LIN {X 0,Y 530.243,Z 390.539,A -85,B 0,C 180,E1 24517.422,E2 24517.422} C_VEL
LIN {X 0,Y 522.245,Z 380.137,A -85,B 0,C 180,E1 24516.068,E2 24516.068} C_VEL
LIN {X 0,Y 518.411,Z 375.142,A -85,B 0,C 180,E1 24515.388,E2 24515.388} C_VEL
LIN {X 0,Y 515.16,Z 370.904,A -85,B 0,C 180,E1 24514.795,E2 24514.795} C_VEL
LIN {X 0,Y 511.277,Z 366.368,A -85,B 0,C 180,E1 24514.077,E2 24514.077} C_VEL
LIN {X 0,Y 510.058,Z 364.29,A -85,B 0,C 180,E1 24513.831,E2 24513.831} C_VEL
LIN {X 0,Y 507.318,Z 361.986,A -85,B 0,C 180,E1 24513.326,E2 24513.326} C_VEL
LIN {X 0,Y 505.948,Z 358.981,A -85,B 0,C 180,E1 24513.023,E2 24513.023} C_VEL
LIN {X 0,Y 505.819,Z 358.226,A -85,B 0,C 180,E1 24512.977,E2 24512.977} C_VEL
LIN {X 0,Y 505.821,Z 358.219,A -85,B 0,C 180,E1 24509.486,E2 24509.486} C_VEL
LIN {X 0,Y 505.867,Z 358.21,A -85,B 0,C 180,E1 24506.154,E2 24506.154} C_VEL
LIN {X 0,Y 505.817,Z 358.219,A -85,B 0,C 180,E1 24502.796,E2 24502.796} C_VEL
LIN {X 0,Y 505.818,Z 358.222,A -85,B 0,C 180,E1 24499.276,E2 24499.276} C_VEL
LIN {X 0,Y 505.867,Z 358.218,A -85,B 0,C 180,E1 24495.829,E2 24495.829} C_VEL
LIN {X 0,Y 505.827,Z 358.218,A -85,B 0,C 180,E1 24492.443,E2 24492.443} C_VEL
LIN {X 0,Y 505.81,Z 358.211,A -85,B 0,C 180,E1 24488.985,E2 24488.985} C_VEL
LIN {X 0,Y 505.861,Z 358.197,A -85,B 0,C 180,E1 24485.672,E2 24485.672} C_VEL
LIN {X 0,Y 505.825,Z 358.208,A -85,B 0,C 180,E1 24482.266,E2 24482.266} C_VEL
LIN {X 0,Y 505.814,Z 358.223,A -85,B 0,C 180,E1 24478.867,E2 24478.867} C_VEL
LIN {X 0,Y 505.86,Z 358.216,A -85,B 0,C 180,E1 24475.465,E2 24475.465} C_VEL
LIN {X 0,Y 505.819,Z 358.203,A -85,B 0,C 180,E1 24472.161,E2 24472.161} C_VEL
LIN {X 0,Y 505.809,Z 358.199,A -85,B 0,C 180,E1 24468.666,E2 24468.666} C_VEL
LIN {X 0,Y 505.856,Z 358.198,A -85,B 0,C 180,E1 24465.227,E2 24465.227} C_VEL
LIN {X 0,Y 505.836,Z 358.211,A -85,B 0,C 180,E1 24461.801,E2 24461.801} C_VEL
LIN {X 0,Y 505.811,Z 358.223,A -85,B 0,C 180,E1 24458.427,E2 24458.427} C_VEL
LIN {X 0,Y 505.86,Z 358.216,A -85,B 0,C 180,E1 24455.101,E2 24455.101} C_VEL
LIN {X 0,Y 505.833,Z 358.216,A -85,B 0,C 180,E1 24451.679,E2 24451.679} C_VEL
LIN {X 0,Y 505.809,Z 358.224,A -85,B 0,C 180,E1 24448.215,E2 24448.215} C_VEL
LIN {X 0,Y 505.856,Z 358.329,A -85,B 0,C 180,E1 24446.764,E2 24446.764} C_VEL
LIN {X 0,Y 507.026,Z 361.574,A -85,B 0,C 180,E1 24446.076,E2 24446.076} C_VEL
LIN {X 0,Y 508.127,Z 363.457,A -85,B 0,C 180,E1 24445.614,E2 24445.614} C_VEL
LIN {X 0,Y 511.472,Z 370.526,A -85,B 0,C 180,E1 24444.127,E2 24444.127} C_VEL
LIN {X 0,Y 517.191,Z 378.321,A -85,B 0,C 180,E1 24443.057,E2 24443.057} C_VEL
LIN {X 0,Y 526.687,Z 391.502,A -85,B 0,C 180,E1 24441.382,E2 24441.382} C_VEL
LIN {X 0,Y 538.736,Z 409.397,A -85,B 0,C 180,E1 24439.401,E2 24439.401} C_VEL
LIN {X 0,Y 550.421,Z 428.049,A -85,B 0,C 180,E1 24437.609,E2 24437.609} C_VEL
LIN {X 0,Y 559.833,Z 444.357,A -85,B 0,C 180,E1 24436.239,E2 24436.239} C_VEL
LIN {X 0,Y 551.218,Z 697.847,A -85,B 0,C 180,E1 24432.584,E2 24432.584} C_VEL
LIN {X 0,Y 548.851,Z 765.211,A -85,B 0,C 180,E1 24431.594,E2 24431.594} C_VEL
LIN {X 0,Y 546.947,Z 790.534,A -85,B 0,C 180,E1 24431.062,E2 24431.062} C_VEL
LIN {X 0,Y 544.812,Z 812.3,A -85,B 0,C 180,E1 24430.449,E2 24430.449} C_VEL
LIN {X 0,Y 541.812,Z 837.253,A -85,B 0,C 180,E1 24429.545,E2 24429.545} C_VEL
LIN {X 0,Y 538.992,Z 857.715,A -85,B 0,C 180,E1 24428.627,E2 24428.627} C_VEL
LIN {X 0,Y 535.358,Z 881.083,A -85,B 0,C 180,E1 24427.373,E2 24427.373} C_VEL
LIN {X 0,Y 532.124,Z 900.104,A -85,B 0,C 180,E1 24426.159,E2 24426.159} C_VEL
LIN {X 0,Y 528.453,Z 920.63,A -85,B 0,C 180,E1 24424.651,E2 24424.651} C_VEL
LIN {X 0,Y 524.681,Z 940.175,A -85,B 0,C 180,E1 24422.962,E2 24422.962} C_VEL
LIN {X 0,Y 521.204,Z 958.071,A -85,B 0,C 180,E1 24421.196,E2 24421.196} C_VEL
LIN {X 0,Y 517.662,Z 976.147,A -85,B 0,C 180,E1 24419.127,E2 24419.127} C_VEL
LIN {X 0,Y 514.766,Z 991.223,A -85,B 0,C 180,E1 24417.159,E2 24417.159} C_VEL
LIN {X 0,Y 511.753,Z 1007.595,A -85,B 0,C 180,E1 24414.695,E2 24414.695} C_VEL
LIN {X 0,Y 509.578,Z 1020.26,A -85,B 0,C 180,E1 24412.497,E2 24412.497} C_VEL
LIN {X 0,Y 507.526,Z 1033.62,A -85,B 0,C 180,E1 24409.808,E2 24409.808} C_VEL
LIN {X 0,Y 506.184,Z 1043.698,A -85,B 0,C 180,E1 24407.427,E2 24407.427} C_VEL
LIN {X 0,Y 505.112,Z 1053.565,A -85,B 0,C 180,E1 24404.678,E2 24404.678} C_VEL
LIN {X 0,Y 504.506,Z 1060.698,A -85,B 0,C 180,E1 24402.243,E2 24402.243} C_VEL
LIN {X 0,Y 504.146,Z 1066.814,A -85,B 0,C 180,E1 24399.693,E2 24399.693} C_VEL
LIN {X 0,Y 503.971,Z 1071.694,A -85,B 0,C 180,E1 24396.951,E2 24396.951} C_VEL
LIN {X 0,Y 503.931,Z 1074.534,A -85,B 0,C 180,E1 24394.666,E2 24394.666} C_VEL
LIN {X 0,Y 503.925,Z 1076.418,A -85,B 0,C 180,E1 24392.161,E2 24392.161} C_VEL
LIN {X 0,Y 503.916,Z 1076.851,A -85,B 0,C 180,E1 24389.432,E2 24389.432} C_VEL
LIN {X 0,Y 503.926,Z 1076.004,A -85,B 0,C 180,E1 24387.157,E2 24387.157} C_VEL
LIN {X 0,Y 503.939,Z 1073.839,A -85,B 0,C 180,E1 24384.649,E2 24384.649} C_VEL
LIN {X 0,Y 504.022,Z 1069.764,A -85,B 0,C 180,E1 24381.863,E2 24381.863} C_VEL
LIN {X 0,Y 504.23,Z 1064.959,A -85,B 0,C 180,E1 24379.488,E2 24379.488} C_VEL
LIN {X 0,Y 504.701,Z 1058.167,A -85,B 0,C 180,E1 24376.831,E2 24376.831} C_VEL
LIN {X 0,Y 505.456,Z 1049.904,A -85,B 0,C 180,E1 24374.276,E2 24374.276} C_VEL
LIN {X 0,Y 506.477,Z 1041.045,A -85,B 0,C 180,E1 24371.944,E2 24371.944} C_VEL
LIN {X 0,Y 508.133,Z 1028.955,A -85,B 0,C 180,E1 24369.256,E2 24369.256} C_VEL
LIN {X 0,Y 509.968,Z 1017.316,A -85,B 0,C 180,E1 24367.034,E2 24367.034} C_VEL
LIN {X 0,Y 512.628,Z 1001.746,A -85,B 0,C 180,E1 24364.465,E2 24364.465} C_VEL
LIN {X 0,Y 515.141,Z 987.899,A -85,B 0,C 180,E1 24362.486,E2 24362.486} C_VEL
LIN {X 0,Y 518.363,Z 970.778,A -85,B 0,C 180,E1 24360.333,E2 24360.333} C_VEL
LIN {X 0,Y 521.652,Z 953.358,A -85,B 0,C 180,E1 24358.448,E2 24358.448} C_VEL
LIN {X 0,Y 525.288,Z 934.182,A -85,B 0,C 180,E1 24356.625,E2 24356.625} C_VEL
LIN {X 0,Y 528.894,Z 913.938,A -85,B 0,C 180,E1 24354.986,E2 24354.986} C_VEL
LIN {X 0,Y 532.482,Z 893.313,A -85,B 0,C 180,E1 24353.536,E2 24353.536} C_VEL
LIN {X 0,Y 535.856,Z 871.76,A -85,B 0,C 180,E1 24352.263,E2 24352.263} C_VEL
LIN {X 0,Y 539.01,Z 850.159,A -85,B 0,C 180,E1 24351.181,E2 24351.181} C_VEL
LIN {X 0,Y 541.922,Z 826.849,A -85,B 0,C 180,E1 24350.224,E2 24350.224} C_VEL
LIN {X 0,Y 544.113,Z 806.615,A -85,B 0,C 180,E1 24349.551,E2 24349.551} C_VEL
LIN {X 0,Y 546.315,Z 781.962,A -85,B 0,C 180,E1 24348.911,E2 24348.911} C_VEL
LIN {X 0,Y 547.686,Z 758.897,A -85,B 0,C 180,E1 24348.481,E2 24348.481} C_VEL
LIN {X 0,Y 555.231,Z 521.007,A -85,B 0,C 180,E1 24345.07,E2 24345.07} C_VEL
LIN {X 0,Y 557.675,Z 443.181,A -85,B 0,C 180,E1 24343.938,E2 24343.938} C_VEL
LIN {X 0,Y 544.63,Z 420.749,A -85,B 0,C 180,E1 24342.125,E2 24342.125} C_VEL
LIN {X 0,Y 532.554,Z 401.419,A -85,B 0,C 180,E1 24340.338,E2 24340.338} C_VEL
LIN {X 0,Y 522.976,Z 387.268,A -85,B 0,C 180,E1 24338.838,E2 24338.838} C_VEL
LIN {X 0,Y 514.362,Z 375.002,A -85,B 0,C 180,E1 24337.408,E2 24337.408} C_VEL
LIN {X 0,Y 511.191,Z 370.226,A -85,B 0,C 180,E1 24336.835,E2 24336.835} C_VEL
LIN {X 0,Y 507.157,Z 361.687,A -85,B 0,C 180,E1 24335.095,E2 24335.095} C_VEL
LIN {X 0,Y 505.824,Z 358.204,A -85,B 0,C 180,E1 24334.358,E2 24334.358} C_VEL
LIN {X 0,Y 505.852,Z 358.197,A -85,B 0,C 180,E1 24331.058,E2 24331.058} C_VEL
LIN {X 0,Y 505.811,Z 358.2,A -85,B 0,C 180,E1 24327.674,E2 24327.674} C_VEL
LIN {X 0,Y 505.823,Z 358.203,A -85,B 0,C 180,E1 24324.154,E2 24324.154} C_VEL
LIN {X 0,Y 505.861,Z 358.219,A -85,B 0,C 180,E1 24320.842,E2 24320.842} C_VEL
LIN {X 0,Y 505.814,Z 358.22,A -85,B 0,C 180,E1 24317.367,E2 24317.367} C_VEL
LIN {X 0,Y 505.814,Z 358.199,A -85,B 0,C 180,E1 24313.839,E2 24313.839} C_VEL
LIN {X 0,Y 505.862,Z 358.197,A -85,B 0,C 180,E1 24310.477,E2 24310.477} C_VEL
LIN {X 0,Y 505.823,Z 358.222,A -85,B 0,C 180,E1 24307.04,E2 24307.04} C_VEL
LIN {X 0,Y 505.81,Z 358.202,A -85,B 0,C 180,E1 24303.513,E2 24303.513} C_VEL
LIN {X 0,Y 505.858,Z 358.193,A -85,B 0,C 180,E1 24300.113,E2 24300.113} C_VEL
LIN {X 0,Y 505.833,Z 358.221,A -85,B 0,C 180,E1 24296.714,E2 24296.714} C_VEL
LIN {X 0,Y 505.808,Z 358.199,A -85,B 0,C 180,E1 24293.302,E2 24293.302} C_VEL
LIN {X 0,Y 505.858,Z 358.198,A -85,B 0,C 180,E1 24289.983,E2 24289.983} C_VEL
LIN {X 0,Y 505.837,Z 358.22,A -85,B 0,C 180,E1 24286.511,E2 24286.511} C_VEL
LIN {X 0,Y 505.811,Z 358.202,A -85,B 0,C 180,E1 24283.092,E2 24283.092} C_VEL
LIN {X 0,Y 505.858,Z 358.195,A -85,B 0,C 180,E1 24279.763,E2 24279.763} C_VEL
LIN {X 0,Y 505.829,Z 358.223,A -85,B 0,C 180,E1 24276.465,E2 24276.465} C_VEL
LIN {X 0,Y 505.815,Z 358.223,A -85,B 0,C 180,E1 24272.957,E2 24272.957} C_VEL
LIN {X 0,Y 505.863,Z 358.201,A -85,B 0,C 180,E1 24269.601,E2 24269.601} C_VEL
LIN {X 0,Y 505.831,Z 358.202,A -85,B 0,C 180,E1 24266.257,E2 24266.257} C_VEL
LIN {X 0,Y 505.814,Z 358.208,A -85,B 0,C 180,E1 24262.778,E2 24262.778} C_VEL
LIN {X 0,Y 505.887,Z 358.359,A -85,B 0,C 180,E1 24261.782,E2 24261.782} C_VEL
LIN {X 0,Y 507.038,Z 361.49,A -85,B 0,C 180,E1 24261.537,E2 24261.537} C_VEL
LIN {X 0,Y 509.577,Z 364.042,A -85,B 0,C 180,E1 24261.104,E2 24261.104} C_VEL
LIN {X 0,Y 510.514,Z 365.429,A -85,B 0,C 180,E1 24260.936,E2 24260.936} C_VEL
LIN {X 0,Y 513.243,Z 369.092,A -85,B 0,C 180,E1 24260.463,E2 24260.463} C_VEL
LIN {X 0,Y 514.716,Z 370.731,A -85,B 0,C 180,E1 24260.219,E2 24260.219} C_VEL
LIN {X 0,Y 517.989,Z 375.01,A -85,B 0,C 180,E1 24259.673,E2 24259.673} C_VEL
LIN {X 0,Y 531.008,Z 392.505,A -85,B 0,C 180,E1 24257.614,E2 24257.614} C_VEL
LIN {X 0,Y 543.149,Z 409.924,A -85,B 0,C 180,E1 24255.83,E2 24255.83} C_VEL
LIN {X 0,Y 556.689,Z 432.23,A -85,B 0,C 180,E1 24253.943,E2 24253.943} C_VEL
LIN {X 0,Y 557.876,Z 434.704,A -85,B 0,C 180,E1 24253.775,E2 24253.775} C_VEL
LIN {X 0,Y 549.924,Z 680.488,A -85,B 0,C 180,E1 24250.254,E2 24250.254} C_VEL
LIN {X 0,Y 547.775,Z 743.673,A -85,B 0,C 180,E1 24249.329,E2 24249.329} C_VEL
LIN {X 0,Y 546.096,Z 768.42,A -85,B 0,C 180,E1 24248.795,E2 24248.795} C_VEL
LIN {X 0,Y 544.147,Z 790.154,A -85,B 0,C 180,E1 24248.172,E2 24248.172} C_VEL
LIN {X 0,Y 541.471,Z 814.447,A -85,B 0,C 180,E1 24247.278,E2 24247.278} C_VEL
LIN {X 0,Y 538.798,Z 834.992,A -85,B 0,C 180,E1 24246.35,E2 24246.35} C_VEL
LIN {X 0,Y 535.419,Z 857.913,A -85,B 0,C 180,E1 24245.113,E2 24245.113} C_VEL
LIN {X 0,Y 535.072,Z 860.018,A -85,B 0,C 180,E1 24244.984,E2 24244.984} C_VEL
LIN {X 0,Y 533.151,Z 866.91,A -85,B 0,C 180,E1 24244.627,E2 24244.627} C_VEL
LIN {X 0,Y 525.296,Z 883.992,A -85,B 0,C 180,E1 24243.86,E2 24243.86} C_VEL
LIN {X 0,Y 523.292,Z 890.316,A -85,B 0,C 180,E1 24243.44,E2 24243.44} C_VEL
LIN {X 0,Y 519.831,Z 908.643,A -85,B 0,C 180,E1 24241.935,E2 24241.935} C_VEL
LIN {X 0,Y 515.922,Z 928.193,A -85,B 0,C 180,E1 24240.069,E2 24240.069} C_VEL
LIN {X 0,Y 512.604,Z 944.372,A -85,B 0,C 180,E1 24238.294,E2 24238.294} C_VEL
LIN {X 0,Y 508.891,Z 962.559,A -85,B 0,C 180,E1 24235.986,E2 24235.986} C_VEL
LIN {X 0,Y 506.164,Z 976.066,A -85,B 0,C 180,E1 24234.013,E2 24234.013} C_VEL
LIN {X 0,Y 503.35,Z 990.707,A -85,B 0,C 180,E1 24231.561,E2 24231.561} C_VEL
LIN {X 0,Y 501.164,Z 1002.678,A -85,B 0,C 180,E1 24229.22,E2 24229.22} C_VEL
LIN {X 0,Y 499.344,Z 1014.112,A -85,B 0,C 180,E1 24226.639,E2 24226.639} C_VEL
LIN {X 0,Y 497.986,Z 1023.606,A -85,B 0,C 180,E1 24224.061,E2 24224.061} C_VEL
LIN {X 0,Y 497.066,Z 1031.627,A -85,B 0,C 180,E1 24221.487,E2 24221.487} C_VEL
LIN {X 0,Y 496.434,Z 1038.548,A -85,B 0,C 180,E1 24218.688,E2 24218.688} C_VEL
LIN {X 0,Y 496.146,Z 1043.064,A -85,B 0,C 180,E1 24216.364,E2 24216.364} C_VEL
LIN {X 0,Y 495.985,Z 1047.067,A -85,B 0,C 180,E1 24213.583,E2 24213.583} C_VEL
LIN {X 0,Y 495.938,Z 1049.294,A -85,B 0,C 180,E1 24210.924,E2 24210.924} C_VEL
LIN {X 0,Y 495.918,Z 1050.148,A -85,B 0,C 180,E1 24208.614,E2 24208.614} C_VEL
LIN {X 0,Y 495.936,Z 1049.805,A -85,B 0,C 180,E1 24205.838,E2 24205.838} C_VEL
LIN {X 0,Y 495.968,Z 1048.022,A -85,B 0,C 180,E1 24203.285,E2 24203.285} C_VEL
LIN {X 0,Y 496.06,Z 1045.155,A -85,B 0,C 180,E1 24200.837,E2 24200.837} C_VEL
LIN {X 0,Y 496.332,Z 1040.111,A -85,B 0,C 180,E1 24197.906,E2 24197.906} C_VEL
LIN {X 0,Y 496.805,Z 1034.416,A -85,B 0,C 180,E1 24195.429,E2 24195.429} C_VEL
LIN {X 0,Y 497.664,Z 1026.716,A -85,B 0,C 180,E1 24192.701,E2 24192.701} C_VEL
LIN {X 0,Y 498.91,Z 1017.376,A -85,B 0,C 180,E1 24190.043,E2 24190.043} C_VEL
LIN {X 0,Y 500.649,Z 1006.723,A -85,B 0,C 180,E1 24187.452,E2 24187.452} C_VEL
LIN {X 0,Y 502.833,Z 994.441,A -85,B 0,C 180,E1 24184.941,E2 24184.941} C_VEL
LIN {X 0,Y 505.349,Z 981.711,A -85,B 0,C 180,E1 24182.673,E2 24182.673} C_VEL
LIN {X 0,Y 508.518,Z 966.224,A -85,B 0,C 180,E1 24180.297,E2 24180.297} C_VEL
LIN {X 0,Y 511.718,Z 951.187,A -85,B 0,C 180,E1 24178.29,E2 24178.29} C_VEL
LIN {X 0,Y 515.692,Z 932.365,A -85,B 0,C 180,E1 24176.114,E2 24176.114} C_VEL
LIN {X 0,Y 519.195,Z 915.589,A -85,B 0,C 180,E1 24174.436,E2 24174.436} C_VEL
LIN {X 0,Y 523.484,Z 894.286,A -85,B 0,C 180,E1 24172.598,E2 24172.598} C_VEL
LIN {X 0,Y 526.959,Z 875.808,A -85,B 0,C 180,E1 24171.232,E2 24171.232} C_VEL
LIN {X 0,Y 530.668,Z 854.628,A -85,B 0,C 180,E1 24169.879,E2 24169.879} C_VEL
LIN {X 0,Y 533.938,Z 833.645,A -85,B 0,C 180,E1 24168.763,E2 24168.763} C_VEL
LIN {X 0,Y 537.103,Z 810.848,A -85,B 0,C 180,E1 24167.738,E2 24167.738} C_VEL
LIN {X 0,Y 539.796,Z 787.034,A -85,B 0,C 180,E1 24166.895,E2 24166.895} C_VEL
LIN {X 0,Y 542.027,Z 763.422,A -85,B 0,C 180,E1 24166.239,E2 24166.239} C_VEL
LIN {X 0,Y 543.601,Z 738.929,A -85,B 0,C 180,E1 24165.755,E2 24165.755} C_VEL
LIN {X 0,Y 552.114,Z 499.336,A -85,B 0,C 180,E1 24162.264,E2 24162.264} C_VEL
LIN {X 0,Y 554.239,Z 438.354,A -85,B 0,C 180,E1 24161.36,E2 24161.36} C_VEL
LIN {X 0,Y 541.092,Z 417.091,A -85,B 0,C 180,E1 24159.385,E2 24159.385} C_VEL
LIN {X 0,Y 530.106,Z 401.533,A -85,B 0,C 180,E1 24157.637,E2 24157.637} C_VEL
LIN {X 0,Y 519.296,Z 387.153,A -85,B 0,C 180,E1 24155.793,E2 24155.793} C_VEL
LIN {X 0,Y 514.694,Z 381.339,A -85,B 0,C 180,E1 24154.966,E2 24154.966} C_VEL
LIN {X 0,Y 510.833,Z 376.392,A -85,B 0,C 180,E1 24154.246,E2 24154.246} C_VEL
LIN {X 0,Y 507.61,Z 372.243,A -85,B 0,C 180,E1 24153.626,E2 24153.626} C_VEL
LIN {X 0,Y 506.536,Z 370.989,A -85,B 0,C 180,E1 24153.418,E2 24153.418} C_VEL
LIN {X 0,Y 503.64,Z 367.828,A -85,B 0,C 180,E1 24152.854,E2 24152.854} C_VEL
LIN {X 0,Y 502.365,Z 365.417,A -85,B 0,C 180,E1 24152.575,E2 24152.575} C_VEL
LIN {X 0,Y 499.464,Z 363.017,A -85,B 0,C 180,E1 24152.006,E2 24152.006} C_VEL
LIN {X 0,Y 498.07,Z 360.156,A -85,B 0,C 180,E1 24151.683,E2 24151.683} C_VEL
LIN {X 0,Y 497.886,Z 359.196,A -85,B 0,C 180,E1 24151.612,E2 24151.612} C_VEL
LIN {X 0,Y 497.942,Z 359.189,A -85,B 0,C 180,E1 24148.172,E2 24148.172} C_VEL
LIN {X 0,Y 497.886,Z 359.195,A -85,B 0,C 180,E1 24144.691,E2 24144.691} C_VEL
LIN {X 0,Y 497.874,Z 359.195,A -85,B 0,C 180,E1 24141.192,E2 24141.192} C_VEL
LIN {X 0,Y 497.913,Z 359.189,A -85,B 0,C 180,E1 24137.773,E2 24137.773} C_VEL
LIN {X 0,Y 497.889,Z 359.193,A -85,B 0,C 180,E1 24134.42,E2 24134.42} C_VEL
LIN {X 0,Y 497.873,Z 359.204,A -85,B 0,C 180,E1 24130.999,E2 24130.999} C_VEL
LIN {X 0,Y 497.92,Z 359.208,A -85,B 0,C 180,E1 24127.616,E2 24127.616} C_VEL
LIN {X 0,Y 497.899,Z 359.204,A -85,B 0,C 180,E1 24124.146,E2 24124.146} C_VEL
LIN {X 0,Y 497.869,Z 359.195,A -85,B 0,C 180,E1 24120.69,E2 24120.69} C_VEL
LIN {X 0,Y 497.905,Z 359.186,A -85,B 0,C 180,E1 24117.353,E2 24117.353} C_VEL
LIN {X 0,Y 497.906,Z 359.195,A -85,B 0,C 180,E1 24113.89,E2 24113.89} C_VEL
LIN {X 0,Y 497.871,Z 359.213,A -85,B 0,C 180,E1 24110.521,E2 24110.521} C_VEL
LIN {X 0,Y 497.892,Z 359.209,A -85,B 0,C 180,E1 24107.002,E2 24107.002} C_VEL
LIN {X 0,Y 497.908,Z 359.189,A -85,B 0,C 180,E1 24103.671,E2 24103.671} C_VEL
LIN {X 0,Y 497.868,Z 359.188,A -85,B 0,C 180,E1 24100.281,E2 24100.281} C_VEL
LIN {X 0,Y 497.89,Z 359.187,A -85,B 0,C 180,E1 24096.82,E2 24096.82} C_VEL
LIN {X 0,Y 497.924,Z 359.186,A -85,B 0,C 180,E1 24093.331,E2 24093.331} C_VEL
LIN {X 0,Y 497.876,Z 359.211,A -85,B 0,C 180,E1 24089.949,E2 24089.949} C_VEL
LIN {X 0,Y 497.886,Z 359.31,A -85,B 0,C 180,E1 24088.023,E2 24088.023} C_VEL
LIN {X 0,Y 499.189,Z 362.632,A -85,B 0,C 180,E1 24087.26,E2 24087.26} C_VEL
LIN {X 0,Y 500.218,Z 364.49,A -85,B 0,C 180,E1 24086.79,E2 24086.79} C_VEL
LIN {X 0,Y 502.776,Z 369.865,A -85,B 0,C 180,E1 24085.577,E2 24085.577} C_VEL
LIN {X 0,Y 513.514,Z 384.325,A -85,B 0,C 180,E1 24083.48,E2 24083.48} C_VEL
LIN {X 0,Y 523.228,Z 398.04,A -85,B 0,C 180,E1 24081.727,E2 24081.727} C_VEL
LIN {X 0,Y 534.82,Z 415.4,A -85,B 0,C 180,E1 24079.781,E2 24079.781} C_VEL
LIN {X 0,Y 546.385,Z 434.053,A -85,B 0,C 180,E1 24077.969,E2 24077.969} C_VEL
LIN {X 0,Y 554.244,Z 447.991,A -85,B 0,C 180,E1 24076.792,E2 24076.792} C_VEL
LIN {X 0,Y 545.342,Z 699.596,A -85,B 0,C 180,E1 24073.135,E2 24073.135} C_VEL
LIN {X 0,Y 542.94,Z 765.137,A -85,B 0,C 180,E1 24072.163,E2 24072.163} C_VEL
LIN {X 0,Y 540.977,Z 790.404,A -85,B 0,C 180,E1 24071.628,E2 24071.628} C_VEL
LIN {X 0,Y 538.79,Z 811.938,A -85,B 0,C 180,E1 24071.02,E2 24071.02} C_VEL
LIN {X 0,Y 535.62,Z 837.328,A -85,B 0,C 180,E1 24070.094,E2 24070.094} C_VEL
LIN {X 0,Y 532.72,Z 857.586,A -85,B 0,C 180,E1 24069.178,E2 24069.178} C_VEL
LIN {X 0,Y 528.916,Z 881.067,A -85,B 0,C 180,E1 24067.908,E2 24067.908} C_VEL
LIN {X 0,Y 525.437,Z 900.712,A -85,B 0,C 180,E1 24066.639,E2 24066.639} C_VEL
LIN {X 0,Y 521.595,Z 921.255,A -85,B 0,C 180,E1 24065.106,E2 24065.106} C_VEL
LIN {X 0,Y 517.677,Z 940.697,A -85,B 0,C 180,E1 24063.4,E2 24063.4} C_VEL
LIN {X 0,Y 513.853,Z 959.576,A -85,B 0,C 180,E1 24061.504,E2 24061.504} C_VEL
LIN {X 0,Y 510.258,Z 976.954,A -85,B 0,C 180,E1 24059.463,E2 24059.463} C_VEL
LIN {X 0,Y 506.928,Z 993.639,A -85,B 0,C 180,E1 24057.233,E2 24057.233} C_VEL
LIN {X 0,Y 503.991,Z 1008.732,A -85,B 0,C 180,E1 24054.872,E2 24054.872} C_VEL
LIN {X 0,Y 501.516,Z 1022.662,A -85,B 0,C 180,E1 24052.383,E2 24052.383} C_VEL
LIN {X 0,Y 499.522,Z 1035.008,A -85,B 0,C 180,E1 24049.773,E2 24049.773} C_VEL
LIN {X 0,Y 498.083,Z 1045.661,A -85,B 0,C 180,E1 24047.163,E2 24047.163} C_VEL
LIN {X 0,Y 497.047,Z 1054.808,A -85,B 0,C 180,E1 24044.445,E2 24044.445} C_VEL
LIN {X 0,Y 496.461,Z 1061.733,A -85,B 0,C 180,E1 24041.973,E2 24041.973} C_VEL
LIN {X 0,Y 496.072,Z 1068.23,A -85,B 0,C 180,E1 24039.012,E2 24039.012} C_VEL
LIN {X 0,Y 495.952,Z 1072.14,A -85,B 0,C 180,E1 24036.599,E2 24036.599} C_VEL
LIN {X 0,Y 495.92,Z 1075.135,A -85,B 0,C 180,E1 24033.931,E2 24033.931} C_VEL
LIN {X 0,Y 495.924,Z 1076.499,A -85,B 0,C 180,E1 24031.271,E2 24031.271} C_VEL
LIN {X 0,Y 495.93,Z 1076.545,A -85,B 0,C 180,E1 24028.96,E2 24028.96} C_VEL
LIN {X 0,Y 495.924,Z 1075.362,A -85,B 0,C 180,E1 24026.405,E2 24026.405} C_VEL
LIN {X 0,Y 495.952,Z 1072.445,A -85,B 0,C 180,E1 24023.634,E2 24023.634} C_VEL
LIN {X 0,Y 496.055,Z 1068.768,A -85,B 0,C 180,E1 24021.305,E2 24021.305} C_VEL
LIN {X 0,Y 496.357,Z 1063.169,A -85,B 0,C 180,E1 24018.614,E2 24018.614} C_VEL
LIN {X 0,Y 496.943,Z 1055.708,A -85,B 0,C 180,E1 24015.89,E2 24015.89} C_VEL
LIN {X 0,Y 497.799,Z 1047.592,A -85,B 0,C 180,E1 24013.428,E2 24013.428} C_VEL
LIN {X 0,Y 499.241,Z 1036.445,A -85,B 0,C 180,E1 24010.619,E2 24010.619} C_VEL
LIN {X 0,Y 500.875,Z 1025.768,A -85,B 0,C 180,E1 24008.327,E2 24008.327} C_VEL
LIN {X 0,Y 503.406,Z 1010.951,A -85,B 0,C 180,E1 24005.598,E2 24005.598} C_VEL
LIN {X 0,Y 505.876,Z 997.537,A -85,B 0,C 180,E1 24003.468,E2 24003.468} C_VEL
LIN {X 0,Y 509.269,Z 980.036,A -85,B 0,C 180,E1 24001.055,E2 24001.055} C_VEL
LIN {X 0,Y 512.399,Z 964.186,A -85,B 0,C 180,E1 23999.162,E2 23999.162} C_VEL
LIN {X 0,Y 516.202,Z 944.946,A -85,B 0,C 180,E1 23997.155,E2 23997.155} C_VEL
LIN {X 0,Y 519.647,Z 927.057,A -85,B 0,C 180,E1 23995.549,E2 23995.549} C_VEL
LIN {X 0,Y 523.461,Z 906.852,A -85,B 0,C 180,E1 23993.962,E2 23993.962} C_VEL
LIN {X 0,Y 527.087,Z 885.661,A -85,B 0,C 180,E1 23992.556,E2 23992.556} C_VEL
LIN {X 0,Y 530.399,Z 865.227,A -85,B 0,C 180,E1 23991.392,E2 23991.392} C_VEL
LIN {X 0,Y 533.687,Z 841.975,A -85,B 0,C 180,E1 23990.292,E2 23990.292} C_VEL
LIN {X 0,Y 536.298,Z 821.174,A -85,B 0,C 180,E1 23989.482,E2 23989.482} C_VEL
LIN {X 0,Y 539.015,Z 795.008,A -85,B 0,C 180,E1 23988.68,E2 23988.68} C_VEL
LIN {X 0,Y 540.805,Z 772.952,A -85,B 0,C 180,E1 23988.178,E2 23988.178} C_VEL
LIN {X 0,Y 542.31,Z 740.397,A -85,B 0,C 180,E1 23987.651,E2 23987.651} C_VEL
LIN {X 0,Y 550.562,Z 489.738,A -85,B 0,C 180,E1 23984.039,E2 23984.039} C_VEL
LIN {X 0,Y 551.919,Z 446.519,A -85,B 0,C 180,E1 23983.397,E2 23983.397} C_VEL
LIN {X 0,Y 538.465,Z 423.266,A -85,B 0,C 180,E1 23981.47,E2 23981.47} C_VEL
LIN {X 0,Y 525.532,Z 402.827,A -85,B 0,C 180,E1 23979.491,E2 23979.491} C_VEL
LIN {X 0,Y 514.351,Z 386.33,A -85,B 0,C 180,E1 23977.655,E2 23977.655} C_VEL
LIN {X 0,Y 506.757,Z 375.71,A -85,B 0,C 180,E1 23976.33,E2 23976.33} C_VEL
LIN {X 0,Y 502.476,Z 369.783,A -85,B 0,C 180,E1 23975.523,E2 23975.523} C_VEL
LIN {X 0,Y 500.933,Z 366.363,A -85,B 0,C 180,E1 23974.811,E2 23974.811} C_VEL
LIN {X 0,Y 499.417,Z 363.014,A -85,B 0,C 180,E1 23974.097,E2 23974.097} C_VEL
LIN {X 0,Y 497.934,Z 359.493,A -85,B 0,C 180,E1 23973.347,E2 23973.347} C_VEL
LIN {X 0,Y 497.913,Z 359.2,A -85,B 0,C 180,E1 23973.108,E2 23973.108} C_VEL
LIN {X 0,Y 497.87,Z 359.203,A -85,B 0,C 180,E1 23969.74,E2 23969.74} C_VEL
LIN {X 0,Y 497.897,Z 359.191,A -85,B 0,C 180,E1 23966.348,E2 23966.348} C_VEL
LIN {X 0,Y 497.914,Z 359.181,A -85,B 0,C 180,E1 23962.929,E2 23962.929} C_VEL
LIN {X 0,Y 497.868,Z 359.19,A -85,B 0,C 180,E1 23959.597,E2 23959.597} C_VEL
LIN {X 0,Y 497.892,Z 359.206,A -85,B 0,C 180,E1 23956.09,E2 23956.09} C_VEL
LIN {X 0,Y 497.913,Z 359.2,A -85,B 0,C 180,E1 23952.762,E2 23952.762} C_VEL
LIN {X 0,Y 497.868,Z 359.182,A -85,B 0,C 180,E1 23949.362,E2 23949.362} C_VEL
LIN {X 0,Y 497.889,Z 359.199,A -85,B 0,C 180,E1 23945.879,E2 23945.879} C_VEL
LIN {X 0,Y 497.923,Z 359.202,A -85,B 0,C 180,E1 23942.417,E2 23942.417} C_VEL
LIN {X 0,Y 497.871,Z 359.179,A -85,B 0,C 180,E1 23939.079,E2 23939.079} C_VEL
LIN {X 0,Y 497.877,Z 359.202,A -85,B 0,C 180,E1 23935.508,E2 23935.508} C_VEL
LIN {X 0,Y 497.925,Z 359.201,A -85,B 0,C 180,E1 23932.035,E2 23932.035} C_VEL
LIN {X 0,Y 497.896,Z 359.177,A -85,B 0,C 180,E1 23928.526,E2 23928.526} C_VEL
LIN {X 0,Y 497.872,Z 359.2,A -85,B 0,C 180,E1 23925.104,E2 23925.104} C_VEL
LIN {X 0,Y 497.905,Z 359.211,A -85,B 0,C 180,E1 23921.622,E2 23921.622} C_VEL
LIN {X 0,Y 497.915,Z 359.186,A -85,B 0,C 180,E1 23918.191,E2 23918.191} C_VEL
LIN {X 0,Y 497.873,Z 359.185,A -85,B 0,C 180,E1 23914.801,E2 23914.801} C_VEL
LIN {X 0,Y 497.894,Z 359.192,A -85,B 0,C 180,E1 23911.316,E2 23911.316} C_VEL
LIN {X 0,Y 497.924,Z 359.199,A -85,B 0,C 180,E1 23907.933,E2 23907.933} C_VEL
LIN {X 0,Y 497.882,Z 359.207,A -85,B 0,C 180,E1 23904.425,E2 23904.425} C_VEL
LIN {X 0,Y 497.896,Z 359.299,A -85,B 0,C 180,E1 23903.002,E2 23903.002} C_VEL
LIN {X 0,Y 498.968,Z 362.349,A -85,B 0,C 180,E1 23902.758,E2 23902.758} C_VEL
LIN {X 0,Y 501.378,Z 364.864,A -85,B 0,C 180,E1 23902.32,E2 23902.32} C_VEL
LIN {X 0,Y 502.405,Z 365.757,A -85,B 0,C 180,E1 23902.14,E2 23902.14} C_VEL
LIN {X 0,Y 504.947,Z 369.663,A -85,B 0,C 180,E1 23901.662,E2 23901.662} C_VEL
LIN {X 0,Y 506.932,Z 371.815,A -85,B 0,C 180,E1 23901.316,E2 23901.316} C_VEL
LIN {X 0,Y 510.263,Z 376.116,A -85,B 0,C 180,E1 23900.733,E2 23900.733} C_VEL
LIN {X 0,Y 522.858,Z 392.793,A -85,B 0,C 180,E1 23898.645,E2 23898.645} C_VEL
LIN {X 0,Y 535.731,Z 410.892,A -85,B 0,C 180,E1 23896.675,E2 23896.675} C_VEL
LIN {X 0,Y 547.57,Z 429.878,A -85,B 0,C 180,E1 23894.96,E2 23894.96} C_VEL
LIN {X 0,Y 552.133,Z 438.039,A -85,B 0,C 180,E1 23894.317,E2 23894.317} C_VEL
LIN {X 0,Y 543.849,Z 683.906,A -85,B 0,C 180,E1 23890.767,E2 23890.767} C_VEL
LIN {X 0,Y 541.705,Z 744.204,A -85,B 0,C 180,E1 23889.874,E2 23889.874} C_VEL
LIN {X 0,Y 539.965,Z 768.829,A -85,B 0,C 180,E1 23889.337,E2 23889.337} C_VEL
LIN {X 0,Y 537.932,Z 790.735,A -85,B 0,C 180,E1 23888.704,E2 23888.704} C_VEL
LIN {X 0,Y 535.138,Z 815.103,A -85,B 0,C 180,E1 23887.796,E2 23887.796} C_VEL
LIN {X 0,Y 532.371,Z 835.618,A -85,B 0,C 180,E1 23886.859,E2 23886.859} C_VEL
LIN {X 0,Y 528.869,Z 858.448,A -85,B 0,C 180,E1 23885.613,E2 23885.613} C_VEL
LIN {X 0,Y 525.676,Z 877.197,A -85,B 0,C 180,E1 23884.397,E2 23884.397} C_VEL
LIN {X 0,Y 523.292,Z 890.316,A -85,B 0,C 180,E1 23883.44,E2 23883.44} C_VEL
LIN {X 0,Y 521.282,Z 896.832,A -85,B 0,C 180,E1 23883.003,E2 23883.003} C_VEL
LIN {X 0,Y 512.667,Z 913.711,A -85,B 0,C 180,E1 23881.949,E2 23881.949} C_VEL
LIN {X 0,Y 510.97,Z 918.726,A -85,B 0,C 180,E1 23881.516,E2 23881.516} C_VEL
LIN {X 0,Y 507.086,Z 937.373,A -85,B 0,C 180,E1 23879.59,E2 23879.59} C_VEL
LIN {X 0,Y 503.657,Z 953.259,A -85,B 0,C 180,E1 23877.681,E2 23877.681} C_VEL
LIN {X 0,Y 500.357,Z 968.747,A -85,B 0,C 180,E1 23875.572,E2 23875.572} C_VEL
LIN {X 0,Y 497.255,Z 983.636,A -85,B 0,C 180,E1 23873.211,E2 23873.211} C_VEL
LIN {X 0,Y 494.795,Z 996.031,A -85,B 0,C 180,E1 23870.958,E2 23870.958} C_VEL
LIN {X 0,Y 492.447,Z 1008.915,A -85,B 0,C 180,E1 23868.221,E2 23868.221} C_VEL
LIN {X 0,Y 490.905,Z 1018.463,A -85,B 0,C 180,E1 23865.839,E2 23865.839} C_VEL
LIN {X 0,Y 489.579,Z 1028.107,A -85,B 0,C 180,E1 23862.983,E2 23862.983} C_VEL
LIN {X 0,Y 488.821,Z 1034.962,A -85,B 0,C 180,E1 23860.489,E2 23860.489} C_VEL
LIN {X 0,Y 488.319,Z 1041.057,A -85,B 0,C 180,E1 23857.767,E2 23857.767} C_VEL
LIN {X 0,Y 488.052,Z 1045.64,A -85,B 0,C 180,E1 23854.936,E2 23854.936} C_VEL
LIN {X 0,Y 487.969,Z 1048.417,A -85,B 0,C 180,E1 23852.466,E2 23852.466} C_VEL
LIN {X 0,Y 487.93,Z 1050.187,A -85,B 0,C 180,E1 23849.53,E2 23849.53} C_VEL
LIN {X 0,Y 487.928,Z 1050.326,A -85,B 0,C 180,E1 23847.063,E2 23847.063} C_VEL
LIN {X 0,Y 487.948,Z 1049.337,A -85,B 0,C 180,E1 23844.591,E2 23844.591} C_VEL
LIN {X 0,Y 488.031,Z 1046.594,A -85,B 0,C 180,E1 23841.636,E2 23841.636} C_VEL
LIN {X 0,Y 488.194,Z 1042.91,A -85,B 0,C 180,E1 23839.139,E2 23839.139} C_VEL
LIN {X 0,Y 488.586,Z 1037.768,A -85,B 0,C 180,E1 23836.509,E2 23836.509} C_VEL
LIN {X 0,Y 489.35,Z 1030.375,A -85,B 0,C 180,E1 23833.622,E2 23833.622} C_VEL
LIN {X 0,Y 490.397,Z 1022.49,A -85,B 0,C 180,E1 23831.098,E2 23831.098} C_VEL
LIN {X 0,Y 492.126,Z 1011.581,A -85,B 0,C 180,E1 23828.206,E2 23828.206} C_VEL
LIN {X 0,Y 494.034,Z 1001.182,A -85,B 0,C 180,E1 23825.868,E2 23825.868} C_VEL
LIN {X 0,Y 496.796,Z 987.389,A -85,B 0,C 180,E1 23823.202,E2 23823.202} C_VEL
LIN {X 0,Y 499.621,Z 974.079,A -85,B 0,C 180,E1 23820.994,E2 23820.994} C_VEL
LIN {X 0,Y 503.101,Z 958.378,A -85,B 0,C 180,E1 23818.717,E2 23818.717} C_VEL
LIN {X 0,Y 506.634,Z 942.412,A -85,B 0,C 180,E1 23816.725,E2 23816.725} C_VEL
LIN {X 0,Y 510.604,Z 924.617,A -85,B 0,C 180,E1 23814.774,E2 23814.774} C_VEL
LIN {X 0,Y 514.669,Z 905.302,A -85,B 0,C 180,E1 23812.968,E2 23812.968} C_VEL
LIN {X 0,Y 518.595,Z 886.147,A -85,B 0,C 180,E1 23811.411,E2 23811.411} C_VEL
LIN {X 0,Y 522.625,Z 864.682,A -85,B 0,C 180,E1 23809.933,E2 23809.933} C_VEL
LIN {X 0,Y 525.92,Z 845.573,A -85,B 0,C 180,E1 23808.805,E2 23808.805} C_VEL
LIN {X 0,Y 529.613,Z 821.59,A -85,B 0,C 180,E1 23807.623,E2 23807.623} C_VEL
LIN {X 0,Y 532.123,Z 802.454,A -85,B 0,C 180,E1 23806.845,E2 23806.845} C_VEL
LIN {X 0,Y 534.743,Z 779.457,A -85,B 0,C 180,E1 23806.08,E2 23806.08} C_VEL
LIN {X 0,Y 536.744,Z 755.79,A -85,B 0,C 180,E1 23805.491,E2 23805.491} C_VEL
LIN {X 0,Y 538.049,Z 733.759,A -85,B 0,C 180,E1 23805.085,E2 23805.085} C_VEL
LIN {X 0,Y 547.283,Z 482.875,A -85,B 0,C 180,E1 23801.411,E2 23801.411} C_VEL
LIN {X 0,Y 548.708,Z 441.821,A -85,B 0,C 180,E1 23800.79,E2 23800.79} C_VEL
LIN {X 0,Y 535.529,Z 420.602,A -85,B 0,C 180,E1 23798.752,E2 23798.752} C_VEL
LIN {X 0,Y 523.411,Z 403.652,A -85,B 0,C 180,E1 23796.757,E2 23796.757} C_VEL
LIN {X 0,Y 511.927,Z 388.487,A -85,B 0,C 180,E1 23794.705,E2 23794.705} C_VEL
LIN {X 0,Y 507.19,Z 382.618,A -85,B 0,C 180,E1 23793.81,E2 23793.81} C_VEL
LIN {X 0,Y 503.446,Z 377.826,A -85,B 0,C 180,E1 23793.071,E2 23793.071} C_VEL
LIN {X 0,Y 500.235,Z 374.018,A -85,B 0,C 180,E1 23792.425,E2 23792.425} C_VEL
LIN {X 0,Y 498.921,Z 372.158,A -85,B 0,C 180,E1 23792.147,E2 23792.147} C_VEL
LIN {X 0,Y 495.879,Z 368.896,A -85,B 0,C 180,E1 23791.517,E2 23791.517} C_VEL
LIN {X 0,Y 494.405,Z 366.407,A -85,B 0,C 180,E1 23791.181,E2 23791.181} C_VEL
LIN {X 0,Y 491.612,Z 364.144,A -85,B 0,C 180,E1 23790.596,E2 23790.596} C_VEL
LIN {X 0,Y 490.187,Z 361.183,A -85,B 0,C 180,E1 23790.242,E2 23790.242} C_VEL
LIN {X 0,Y 490,Z 360.194,A -85,B 0,C 180,E1 23790.165,E2 23790.165} C_VEL
LIN {X 0,Y 489.946,Z 360.203,A -85,B 0,C 180,E1 23786.809,E2 23786.809} C_VEL
LIN {X 0,Y 489.937,Z 360.203,A -85,B 0,C 180,E1 23783.197,E2 23783.197} C_VEL
LIN {X 0,Y 489.981,Z 360.199,A -85,B 0,C 180,E1 23779.801,E2 23779.801} C_VEL
LIN {X 0,Y 489.973,Z 360.196,A -85,B 0,C 180,E1 23776.235,E2 23776.235} C_VEL
LIN {X 0,Y 489.933,Z 360.192,A -85,B 0,C 180,E1 23772.853,E2 23772.853} C_VEL
LIN {X 0,Y 489.954,Z 360.179,A -85,B 0,C 180,E1 23769.396,E2 23769.396} C_VEL
LIN {X 0,Y 489.968,Z 360.177,A -85,B 0,C 180,E1 23766.092,E2 23766.092} C_VEL
LIN {X 0,Y 489.934,Z 360.192,A -85,B 0,C 180,E1 23762.573,E2 23762.573} C_VEL
LIN {X 0,Y 489.94,Z 360.201,A -85,B 0,C 180,E1 23758.948,E2 23758.948} C_VEL
LIN {X 0,Y 489.979,Z 360.194,A -85,B 0,C 180,E1 23755.435,E2 23755.435} C_VEL
LIN {X 0,Y 489.951,Z 360.18,A -85,B 0,C 180,E1 23752.023,E2 23752.023} C_VEL
LIN {X 0,Y 489.93,Z 360.176,A -85,B 0,C 180,E1 23748.582,E2 23748.582} C_VEL
LIN {X 0,Y 489.964,Z 360.175,A -85,B 0,C 180,E1 23745.1,E2 23745.1} C_VEL
LIN {X 0,Y 489.974,Z 360.182,A -85,B 0,C 180,E1 23741.609,E2 23741.609} C_VEL
LIN {X 0,Y 489.933,Z 360.199,A -85,B 0,C 180,E1 23738.196,E2 23738.196} C_VEL
LIN {X 0,Y 489.943,Z 360.201,A -85,B 0,C 180,E1 23734.623,E2 23734.623} C_VEL
LIN {X 0,Y 489.992,Z 360.197,A -85,B 0,C 180,E1 23731.077,E2 23731.077} C_VEL
LIN {X 0,Y 490.017,Z 360.424,A -85,B 0,C 180,E1 23729.327,E2 23729.327} C_VEL
LIN {X 0,Y 491.418,Z 363.93,A -85,B 0,C 180,E1 23728.472,E2 23728.472} C_VEL
LIN {X 0,Y 492.392,Z 365.741,A -85,B 0,C 180,E1 23727.994,E2 23727.994} C_VEL
LIN {X 0,Y 494.518,Z 369.645,A -85,B 0,C 180,E1 23727.046,E2 23727.046} C_VEL
LIN {X 0,Y 497.801,Z 374.223,A -85,B 0,C 180,E1 23726.332,E2 23726.332} C_VEL
LIN {X 0,Y 507.638,Z 387.39,A -85,B 0,C 180,E1 23724.336,E2 23724.336} C_VEL
LIN {X 0,Y 516.631,Z 399.971,A -85,B 0,C 180,E1 23722.645,E2 23722.645} C_VEL
LIN {X 0,Y 527.787,Z 416.461,A -85,B 0,C 180,E1 23720.693,E2 23720.693} C_VEL
LIN {X 0,Y 540.338,Z 436.58,A -85,B 0,C 180,E1 23718.652,E2 23718.652} C_VEL
LIN {X 0,Y 548.721,Z 451.316,A -85,B 0,C 180,E1 23717.36,E2 23717.36} C_VEL
LIN {X 0,Y 539.493,Z 702.065,A -85,B 0,C 180,E1 23713.689,E2 23713.689} C_VEL
LIN {X 0,Y 537.078,Z 765.181,A -85,B 0,C 180,E1 23712.743,E2 23712.743} C_VEL
LIN {X 0,Y 535.059,Z 790.28,A -85,B 0,C 180,E1 23712.207,E2 23712.207} C_VEL
LIN {X 0,Y 532.837,Z 811.473,A -85,B 0,C 180,E1 23711.606,E2 23711.606} C_VEL
LIN {X 0,Y 529.672,Z 836.124,A -85,B 0,C 180,E1 23710.709,E2 23710.709} C_VEL
LIN {X 0,Y 526.628,Z 856.667,A -85,B 0,C 180,E1 23709.781,E2 23709.781} C_VEL
LIN {X 0,Y 522.863,Z 879.253,A -85,B 0,C 180,E1 23708.566,E2 23708.566} C_VEL
LIN {X 0,Y 519.029,Z 900.032,A -85,B 0,C 180,E1 23707.222,E2 23707.222} C_VEL
LIN {X 0,Y 515.052,Z 920.507,A -85,B 0,C 180,E1 23705.688,E2 23705.688} C_VEL
LIN {X 0,Y 510.952,Z 940.064,A -85,B 0,C 180,E1 23703.959,E2 23703.959} C_VEL
LIN {X 0,Y 507.093,Z 958.257,A -85,B 0,C 180,E1 23702.121,E2 23702.121} C_VEL
LIN {X 0,Y 503.262,Z 975.902,A -85,B 0,C 180,E1 23700.045,E2 23700.045} C_VEL
LIN {X 0,Y 499.916,Z 991.806,A -85,B 0,C 180,E1 23697.906,E2 23697.906} C_VEL
LIN {X 0,Y 496.763,Z 1007.17,A -85,B 0,C 180,E1 23695.515,E2 23695.515} C_VEL
LIN {X 0,Y 494.443,Z 1019.312,A -85,B 0,C 180,E1 23693.349,E2 23693.349} C_VEL
LIN {X 0,Y 492.101,Z 1032.754,A -85,B 0,C 180,E1 23690.58,E2 23690.58} C_VEL
LIN {X 0,Y 490.58,Z 1042.696,A -85,B 0,C 180,E1 23688.17,E2 23688.17} C_VEL
LIN {X 0,Y 489.408,Z 1052.094,A -85,B 0,C 180,E1 23685.524,E2 23685.524} C_VEL
LIN {X 0,Y 488.611,Z 1060.001,A -85,B 0,C 180,E1 23682.768,E2 23682.768} C_VEL
LIN {X 0,Y 488.21,Z 1065.616,A -85,B 0,C 180,E1 23680.383,E2 23680.383} C_VEL
LIN {X 0,Y 487.988,Z 1070.959,A -85,B 0,C 180,E1 23677.417,E2 23677.417} C_VEL
LIN {X 0,Y 487.94,Z 1074.004,A -85,B 0,C 180,E1 23674.937,E2 23674.937} C_VEL
LIN {X 0,Y 487.927,Z 1075.86,A -85,B 0,C 180,E1 23672.466,E2 23672.466} C_VEL
LIN {X 0,Y 487.924,Z 1076.467,A -85,B 0,C 180,E1 23669.648,E2 23669.648} C_VEL
LIN {X 0,Y 487.93,Z 1075.637,A -85,B 0,C 180,E1 23667.181,E2 23667.181} C_VEL
LIN {X 0,Y 487.941,Z 1073.628,A -85,B 0,C 180,E1 23664.709,E2 23664.709} C_VEL
LIN {X 0,Y 488.035,Z 1069.53,A -85,B 0,C 180,E1 23661.721,E2 23661.721} C_VEL
LIN {X 0,Y 488.264,Z 1064.748,A -85,B 0,C 180,E1 23659.26,E2 23659.26} C_VEL
LIN {X 0,Y 488.784,Z 1058.014,A -85,B 0,C 180,E1 23656.514,E2 23656.514} C_VEL
LIN {X 0,Y 489.667,Z 1049.398,A -85,B 0,C 180,E1 23653.755,E2 23653.755} C_VEL
LIN {X 0,Y 490.902,Z 1040.057,A -85,B 0,C 180,E1 23651.227,E2 23651.227} C_VEL
LIN {X 0,Y 492.69,Z 1028.406,A -85,B 0,C 180,E1 23648.574,E2 23648.574} C_VEL
LIN {X 0,Y 494.724,Z 1016.75,A -85,B 0,C 180,E1 23646.284,E2 23646.284} C_VEL
LIN {X 0,Y 497.688,Z 1001.146,A -85,B 0,C 180,E1 23643.64,E2 23643.64} C_VEL
LIN {X 0,Y 500.61,Z 986.526,A -85,B 0,C 180,E1 23641.502,E2 23641.502} C_VEL
LIN {X 0,Y 504.41,Z 968.165,A -85,B 0,C 180,E1 23639.175,E2 23639.175} C_VEL
LIN {X 0,Y 507.711,Z 952.169,A -85,B 0,C 180,E1 23637.416,E2 23637.416} C_VEL
LIN {X 0,Y 511.658,Z 932.877,A -85,B 0,C 180,E1 23635.557,E2 23635.557} C_VEL
LIN {X 0,Y 515.488,Z 913.172,A -85,B 0,C 180,E1 23633.935,E2 23633.935} C_VEL
LIN {X 0,Y 519.375,Z 892.502,A -85,B 0,C 180,E1 23632.46,E2 23632.46} C_VEL
LIN {X 0,Y 522.872,Z 871.802,A -85,B 0,C 180,E1 23631.218,E2 23631.218} C_VEL
LIN {X 0,Y 525.902,Z 852.464,A -85,B 0,C 180,E1 23630.224,E2 23630.224} C_VEL
LIN {X 0,Y 529.266,Z 827.978,A -85,B 0,C 180,E1 23629.182,E2 23629.182} C_VEL
LIN {X 0,Y 531.66,Z 807.467,A -85,B 0,C 180,E1 23628.483,E2 23628.483} C_VEL
LIN {X 0,Y 533.984,Z 783.875,A -85,B 0,C 180,E1 23627.846,E2 23627.846} C_VEL
LIN {X 0,Y 535.574,Z 759.261,A -85,B 0,C 180,E1 23627.373,E2 23627.373} C_VEL
LIN {X 0,Y 543.706,Z 523.272,A -85,B 0,C 180,E1 23623.931,E2 23623.931} C_VEL
LIN {X 0,Y 546.171,Z 449.822,A -85,B 0,C 180,E1 23622.84,E2 23622.84} C_VEL
LIN {X 0,Y 533.572,Z 427.973,A -85,B 0,C 180,E1 23620.987,E2 23620.987} C_VEL
LIN {X 0,Y 520.585,Z 407.244,A -85,B 0,C 180,E1 23618.944,E2 23618.944} C_VEL
LIN {X 0,Y 507.929,Z 388.602,A -85,B 0,C 180,E1 23616.794,E2 23616.794} C_VEL
LIN {X 0,Y 497.103,Z 373.702,A -85,B 0,C 180,E1 23614.802,E2 23614.802} C_VEL
LIN {X 0,Y 494.207,Z 369.566,A -85,B 0,C 180,E1 23614.226,E2 23614.226} C_VEL
LIN {X 0,Y 492.163,Z 365.3,A -85,B 0,C 180,E1 23613.267,E2 23613.267} C_VEL
LIN {X 0,Y 489.994,Z 360.56,A -85,B 0,C 180,E1 23612.182,E2 23612.182} C_VEL
LIN {X 0,Y 489.934,Z 360.191,A -85,B 0,C 180,E1 23612.048,E2 23612.048} C_VEL
LIN {X 0,Y 489.991,Z 360.186,A -85,B 0,C 180,E1 23608.656,E2 23608.656} C_VEL
LIN {X 0,Y 489.963,Z 360.198,A -85,B 0,C 180,E1 23605.118,E2 23605.118} C_VEL
LIN {X 0,Y 489.931,Z 360.197,A -85,B 0,C 180,E1 23601.679,E2 23601.679} C_VEL
LIN {X 0,Y 489.956,Z 360.176,A -85,B 0,C 180,E1 23598.194,E2 23598.194} C_VEL
LIN {X 0,Y 489.99,Z 360.167,A -85,B 0,C 180,E1 23594.657,E2 23594.657} C_VEL
LIN {X 0,Y 489.941,Z 360.196,A -85,B 0,C 180,E1 23591.179,E2 23591.179} C_VEL
LIN {X 0,Y 489.934,Z 360.198,A -85,B 0,C 180,E1 23587.623,E2 23587.623} C_VEL
LIN {X 0,Y 489.975,Z 360.165,A -85,B 0,C 180,E1 23584.213,E2 23584.213} C_VEL
LIN {X 0,Y 489.962,Z 360.184,A -85,B 0,C 180,E1 23580.702,E2 23580.702} C_VEL
LIN {X 0,Y 489.934,Z 360.201,A -85,B 0,C 180,E1 23577.192,E2 23577.192} C_VEL
LIN {X 0,Y 489.946,Z 360.169,A -85,B 0,C 180,E1 23573.656,E2 23573.656} C_VEL
LIN {X 0,Y 489.983,Z 360.18,A -85,B 0,C 180,E1 23570.248,E2 23570.248} C_VEL
LIN {X 0,Y 489.942,Z 360.199,A -85,B 0,C 180,E1 23566.774,E2 23566.774} C_VEL
LIN {X 0,Y 489.934,Z 360.176,A -85,B 0,C 180,E1 23563.154,E2 23563.154} C_VEL
LIN {X 0,Y 489.973,Z 360.171,A -85,B 0,C 180,E1 23559.701,E2 23559.701} C_VEL
LIN {X 0,Y 489.964,Z 360.195,A -85,B 0,C 180,E1 23556.295,E2 23556.295} C_VEL
LIN {X 0,Y 489.94,Z 360.202,A -85,B 0,C 180,E1 23552.797,E2 23552.797} C_VEL
LIN {X 0,Y 489.957,Z 360.186,A -85,B 0,C 180,E1 23549.323,E2 23549.323} C_VEL
LIN {X 0,Y 489.984,Z 360.179,A -85,B 0,C 180,E1 23545.862,E2 23545.862} C_VEL
LIN {X 0,Y 489.958,Z 360.256,A -85,B 0,C 180,E1 23544.291,E2 23544.291} C_VEL
LIN {X 0,Y 491.007,Z 363.245,A -85,B 0,C 180,E1 23544.038,E2 23544.038} C_VEL
LIN {X 0,Y 493.4,Z 365.788,A -85,B 0,C 180,E1 23543.575,E2 23543.575} C_VEL
LIN {X 0,Y 494.526,Z 366.796,A -85,B 0,C 180,E1 23543.365,E2 23543.365} C_VEL
LIN {X 0,Y 496.989,Z 370.604,A -85,B 0,C 180,E1 23542.874,E2 23542.874} C_VEL
LIN {X 0,Y 499.262,Z 372.917,A -85,B 0,C 180,E1 23542.458,E2 23542.458} C_VEL
LIN {X 0,Y 502.564,Z 377.233,A -85,B 0,C 180,E1 23541.847,E2 23541.847} C_VEL
LIN {X 0,Y 512.006,Z 389.56,A -85,B 0,C 180,E1 23540.185,E2 23540.185} C_VEL
LIN {X 0,Y 523.641,Z 405.343,A -85,B 0,C 180,E1 23538.282,E2 23538.282} C_VEL
LIN {X 0,Y 534.992,Z 421.994,A -85,B 0,C 180,E1 23536.545,E2 23536.545} C_VEL
LIN {X 0,Y 546.448,Z 441.202,A -85,B 0,C 180,E1 23534.872,E2 23534.872} C_VEL
LIN {X 0,Y 537.807,Z 687.67,A -85,B 0,C 180,E1 23531.286,E2 23531.286} C_VEL
LIN {X 0,Y 535.684,Z 744.725,A -85,B 0,C 180,E1 23530.432,E2 23530.432} C_VEL
LIN {X 0,Y 533.884,Z 769.233,A -85,B 0,C 180,E1 23529.892,E2 23529.892} C_VEL
LIN {X 0,Y 531.773,Z 791.218,A -85,B 0,C 180,E1 23529.25,E2 23529.25} C_VEL
LIN {X 0,Y 528.953,Z 814.971,A -85,B 0,C 180,E1 23528.361,E2 23528.361} C_VEL
LIN {X 0,Y 526.187,Z 834.834,A -85,B 0,C 180,E1 23527.451,E2 23527.451} C_VEL
LIN {X 0,Y 522.677,Z 857.192,A -85,B 0,C 180,E1 23526.237,E2 23526.237} C_VEL
LIN {X 0,Y 519.054,Z 877.695,A -85,B 0,C 180,E1 23524.899,E2 23524.899} C_VEL
LIN {X 0,Y 515.255,Z 897.885,A -85,B 0,C 180,E1 23523.377,E2 23523.377} C_VEL
LIN {X 0,Y 511.312,Z 917.088,A -85,B 0,C 180,E1 23521.672,E2 23521.672} C_VEL
LIN {X 0,Y 510.97,Z 918.726,A -85,B 0,C 180,E1 23521.516,E2 23521.516} C_VEL
LIN {X 0,Y 508.908,Z 924.702,A -85,B 0,C 180,E1 23521.001,E2 23521.001} C_VEL
LIN {X 0,Y 500.503,Z 939.528,A -85,B 0,C 180,E1 23519.781,E2 23519.781} C_VEL
LIN {X 0,Y 498.41,Z 944.959,A -85,B 0,C 180,E1 23519.204,E2 23519.204} C_VEL
LIN {X 0,Y 494.435,Z 962.729,A -85,B 0,C 180,E1 23516.895,E2 23516.895} C_VEL
LIN {X 0,Y 491.323,Z 976.784,A -85,B 0,C 180,E1 23514.786,E2 23514.786} C_VEL
LIN {X 0,Y 488.087,Z 992.002,A -85,B 0,C 180,E1 23512.144,E2 23512.144} C_VEL
LIN {X 0,Y 485.71,Z 1003.891,A -85,B 0,C 180,E1 23509.731,E2 23509.731} C_VEL
LIN {X 0,Y 483.54,Z 1016.07,A -85,B 0,C 180,E1 23506.828,E2 23506.828} C_VEL
LIN {X 0,Y 482.208,Z 1024.593,A -85,B 0,C 180,E1 23504.408,E2 23504.408} C_VEL
LIN {X 0,Y 481.157,Z 1032.862,A -85,B 0,C 180,E1 23501.629,E2 23501.629} C_VEL
LIN {X 0,Y 480.498,Z 1039.328,A -85,B 0,C 180,E1 23498.858,E2 23498.858} C_VEL
LIN {X 0,Y 480.163,Z 1043.981,A -85,B 0,C 180,E1 23496.336,E2 23496.336} C_VEL
LIN {X 0,Y 479.987,Z 1047.874,A -85,B 0,C 180,E1 23493.344,E2 23493.344} C_VEL
LIN {X 0,Y 479.945,Z 1049.749,A -85,B 0,C 180,E1 23490.955,E2 23490.955} C_VEL
LIN {X 0,Y 479.923,Z 1050.584,A -85,B 0,C 180,E1 23488.567,E2 23488.567} C_VEL
LIN {X 0,Y 479.94,Z 1050.138,A -85,B 0,C 180,E1 23485.579,E2 23485.579} C_VEL
LIN {X 0,Y 479.981,Z 1048.405,A -85,B 0,C 180,E1 23483.06,E2 23483.06} C_VEL
LIN {X 0,Y 480.088,Z 1045.678,A -85,B 0,C 180,E1 23480.651,E2 23480.651} C_VEL
LIN {X 0,Y 480.404,Z 1040.694,A -85,B 0,C 180,E1 23477.621,E2 23477.621} C_VEL
LIN {X 0,Y 480.947,Z 1035.03,A -85,B 0,C 180,E1 23475.061,E2 23475.061} C_VEL
LIN {X 0,Y 481.928,Z 1027.365,A -85,B 0,C 180,E1 23472.237,E2 23472.237} C_VEL
LIN {X 0,Y 483.383,Z 1017.776,A -85,B 0,C 180,E1 23469.412,E2 23469.412} C_VEL
LIN {X 0,Y 485.367,Z 1006.968,A -85,B 0,C 180,E1 23466.701,E2 23466.701} C_VEL
LIN {X 0,Y 487.847,Z 994.643,A -85,B 0,C 180,E1 23464.115,E2 23464.115} C_VEL
LIN {X 0,Y 490.638,Z 981.902,A -85,B 0,C 180,E1 23461.784,E2 23461.784} C_VEL
LIN {X 0,Y 494.168,Z 966.354,A -85,B 0,C 180,E1 23459.343,E2 23459.343} C_VEL
LIN {X 0,Y 497.539,Z 951.848,A -85,B 0,C 180,E1 23457.358,E2 23457.358} C_VEL
LIN {X 0,Y 501.913,Z 933.015,A -85,B 0,C 180,E1 23455.128,E2 23455.128} C_VEL
LIN {X 0,Y 505.593,Z 916.81,A -85,B 0,C 180,E1 23453.468,E2 23453.468} C_VEL
LIN {X 0,Y 509.926,Z 897.147,A -85,B 0,C 180,E1 23451.711,E2 23451.711} C_VEL
LIN {X 0,Y 513.894,Z 877.606,A -85,B 0,C 180,E1 23450.225,E2 23450.225} C_VEL
LIN {X 0,Y 517.938,Z 856.354,A -85,B 0,C 180,E1 23448.829,E2 23448.829} C_VEL
LIN {X 0,Y 521.615,Z 834.431,A -85,B 0,C 180,E1 23447.639,E2 23447.639} C_VEL
LIN {X 0,Y 524.717,Z 813.622,A -85,B 0,C 180,E1 23446.685,E2 23446.685} C_VEL
LIN {X 0,Y 527.783,Z 789.004,A -85,B 0,C 180,E1 23445.78,E2 23445.78} C_VEL
LIN {X 0,Y 530.012,Z 767.069,A -85,B 0,C 180,E1 23445.15,E2 23445.15} C_VEL
LIN {X 0,Y 531.932,Z 740.911,A -85,B 0,C 180,E1 23444.604,E2 23444.604} C_VEL
LIN {X 0,Y 540.794,Z 510.534,A -85,B 0,C 180,E1 23441.191,E2 23441.191} C_VEL
LIN {X 0,Y 543.236,Z 445.431,A -85,B 0,C 180,E1 23440.211,E2 23440.211} C_VEL
LIN {X 0,Y 530.888,Z 425.495,A -85,B 0,C 180,E1 23438.248,E2 23438.248} C_VEL
LIN {X 0,Y 519.483,Z 409.528,A -85,B 0,C 180,E1 23436.324,E2 23436.324} C_VEL
LIN {X 0,Y 508.649,Z 395.076,A -85,B 0,C 180,E1 23434.345,E2 23434.345} C_VEL
LIN {X 0,Y 503.459,Z 388.623,A -85,B 0,C 180,E1 23433.342,E2 23433.342} C_VEL
LIN {X 0,Y 500.253,Z 384.501,A -85,B 0,C 180,E1 23432.695,E2 23432.695} C_VEL
LIN {X 0,Y 496.742,Z 380.013,A -85,B 0,C 180,E1 23431.965,E2 23431.965} C_VEL
LIN {X 0,Y 492.563,Z 375.092,A -85,B 0,C 180,E1 23431.073,E2 23431.073} C_VEL
LIN {X 0,Y 491.539,Z 373.531,A -85,B 0,C 180,E1 23430.839,E2 23430.839} C_VEL
LIN {X 0,Y 488.465,Z 370.552,A -85,B 0,C 180,E1 23430.168,E2 23430.168} C_VEL
LIN {X 0,Y 486.735,Z 367.519,A -85,B 0,C 180,E1 23429.743,E2 23429.743} C_VEL
LIN {X 0,Y 483.812,Z 365.336,A -85,B 0,C 180,E1 23429.091,E2 23429.091} C_VEL
LIN {X 0,Y 482.264,Z 362.395,A -85,B 0,C 180,E1 23428.684,E2 23428.684} C_VEL
LIN {X 0,Y 482.022,Z 361.171,A -85,B 0,C 180,E1 23428.575,E2 23428.575} C_VEL
LIN {X 0,Y 481.997,Z 361.171,A -85,B 0,C 180,E1 23425.037,E2 23425.037} C_VEL
LIN {X 0,Y 482.013,Z 361.168,A -85,B 0,C 180,E1 23421.541,E2 23421.541} C_VEL
LIN {X 0,Y 482.042,Z 361.165,A -85,B 0,C 180,E1 23418.128,E2 23418.128} C_VEL
LIN {X 0,Y 481.999,Z 361.173,A -85,B 0,C 180,E1 23414.66,E2 23414.66} C_VEL
LIN {X 0,Y 482,Z 361.182,A -85,B 0,C 180,E1 23411.121,E2 23411.121} C_VEL
LIN {X 0,Y 482.043,Z 361.186,A -85,B 0,C 180,E1 23407.629,E2 23407.629} C_VEL
LIN {X 0,Y 482.029,Z 361.182,A -85,B 0,C 180,E1 23404.044,E2 23404.044} C_VEL
LIN {X 0,Y 481.993,Z 361.172,A -85,B 0,C 180,E1 23400.594,E2 23400.594} C_VEL
LIN {X 0,Y 482.002,Z 361.165,A -85,B 0,C 180,E1 23397.027,E2 23397.027} C_VEL
LIN {X 0,Y 482.05,Z 361.162,A -85,B 0,C 180,E1 23393.496,E2 23393.496} C_VEL
LIN {X 0,Y 482.015,Z 361.178,A -85,B 0,C 180,E1 23389.965,E2 23389.965} C_VEL
LIN {X 0,Y 481.994,Z 361.191,A -85,B 0,C 180,E1 23386.443,E2 23386.443} C_VEL
LIN {X 0,Y 482.02,Z 361.181,A -85,B 0,C 180,E1 23382.993,E2 23382.993} C_VEL
LIN {X 0,Y 482.042,Z 361.168,A -85,B 0,C 180,E1 23379.479,E2 23379.479} C_VEL
LIN {X 0,Y 481.994,Z 361.168,A -85,B 0,C 180,E1 23376.138,E2 23376.138} C_VEL
LIN {X 0,Y 482.002,Z 361.168,A -85,B 0,C 180,E1 23372.579,E2 23372.579} C_VEL
LIN {X 0,Y 482.039,Z 361.318,A -85,B 0,C 180,E1 23370.792,E2 23370.792} C_VEL
LIN {X 0,Y 483.265,Z 364.613,A -85,B 0,C 180,E1 23369.953,E2 23369.953} C_VEL
LIN {X 0,Y 484.518,Z 366.617,A -85,B 0,C 180,E1 23369.354,E2 23369.354} C_VEL
LIN {X 0,Y 485.699,Z 369.227,A -85,B 0,C 180,E1 23368.749,E2 23368.749} C_VEL
LIN {X 0,Y 491.205,Z 375.925,A -85,B 0,C 180,E1 23367.493,E2 23367.493} C_VEL
LIN {X 0,Y 495.053,Z 381.243,A -85,B 0,C 180,E1 23366.641,E2 23366.641} C_VEL
LIN {X 0,Y 506.429,Z 396.637,A -85,B 0,C 180,E1 23364.307,E2 23364.307} C_VEL
LIN {X 0,Y 516.502,Z 411.273,A -85,B 0,C 180,E1 23362.407,E2 23362.407} C_VEL
LIN {X 0,Y 527.061,Z 427.405,A -85,B 0,C 180,E1 23360.558,E2 23360.558} C_VEL
LIN {X 0,Y 538.473,Z 446.211,A -85,B 0,C 180,E1 23358.69,E2 23358.69} C_VEL
LIN {X 0,Y 543.243,Z 454.93,A -85,B 0,C 180,E1 23357.936,E2 23357.936} C_VEL
LIN {X 0,Y 533.681,Z 704.967,A -85,B 0,C 180,E1 23354.248,E2 23354.248} C_VEL
LIN {X 0,Y 531.274,Z 765.234,A -85,B 0,C 180,E1 23353.336,E2 23353.336} C_VEL
LIN {X 0,Y 529.199,Z 790.162,A -85,B 0,C 180,E1 23352.799,E2 23352.799} C_VEL
LIN {X 0,Y 526.93,Z 811.121,A -85,B 0,C 180,E1 23352.202,E2 23352.202} C_VEL
LIN {X 0,Y 523.593,Z 836.206,A -85,B 0,C 180,E1 23351.284,E2 23351.284} C_VEL
LIN {X 0,Y 520.443,Z 856.712,A -85,B 0,C 180,E1 23350.35,E2 23350.35} C_VEL
LIN {X 0,Y 516.41,Z 879.898,A -85,B 0,C 180,E1 23349.088,E2 23349.088} C_VEL
LIN {X 0,Y 512.556,Z 900,A -85,B 0,C 180,E1 23347.774,E2 23347.774} C_VEL
LIN {X 0,Y 508.269,Z 921.119,A -85,B 0,C 180,E1 23346.169,E2 23346.169} C_VEL
LIN {X 0,Y 504.207,Z 939.745,A -85,B 0,C 180,E1 23344.504,E2 23344.504} C_VEL
LIN {X 0,Y 500.318,Z 957.3,A -85,B 0,C 180,E1 23342.714,E2 23342.714} C_VEL
LIN {X 0,Y 496.118,Z 975.783,A -85,B 0,C 180,E1 23340.523,E2 23340.523} C_VEL
LIN {X 0,Y 492.794,Z 990.826,A -85,B 0,C 180,E1 23338.478,E2 23338.478} C_VEL
LIN {X 0,Y 489.298,Z 1007.022,A -85,B 0,C 180,E1 23335.933,E2 23335.933} C_VEL
LIN {X 0,Y 486.851,Z 1019.146,A -85,B 0,C 180,E1 23333.737,E2 23333.737} C_VEL
LIN {X 0,Y 484.368,Z 1032.585,A -85,B 0,C 180,E1 23330.924,E2 23330.924} C_VEL
LIN {X 0,Y 482.744,Z 1042.645,A -85,B 0,C 180,E1 23328.442,E2 23328.442} C_VEL
LIN {X 0,Y 481.465,Z 1052.283,A -85,B 0,C 180,E1 23325.663,E2 23325.663} C_VEL
LIN {X 0,Y 480.662,Z 1059.81,A -85,B 0,C 180,E1 23322.983,E2 23322.983} C_VEL
LIN {X 0,Y 480.236,Z 1065.421,A -85,B 0,C 180,E1 23320.558,E2 23320.558} C_VEL
LIN {X 0,Y 479.987,Z 1070.757,A -85,B 0,C 180,E1 23317.541,E2 23317.541} C_VEL
LIN {X 0,Y 479.941,Z 1073.798,A -85,B 0,C 180,E1 23315.02,E2 23315.02} C_VEL
LIN {X 0,Y 479.929,Z 1075.652,A -85,B 0,C 180,E1 23312.508,E2 23312.508} C_VEL
LIN {X 0,Y 479.927,Z 1076.252,A -85,B 0,C 180,E1 23309.642,E2 23309.642} C_VEL
LIN {X 0,Y 479.932,Z 1075.418,A -85,B 0,C 180,E1 23307.134,E2 23307.134} C_VEL
LIN {X 0,Y 479.942,Z 1073.521,A -85,B 0,C 180,E1 23304.74,E2 23304.74} C_VEL
LIN {X 0,Y 480.021,Z 1069.777,A -85,B 0,C 180,E1 23301.857,E2 23301.857} C_VEL
LIN {X 0,Y 480.272,Z 1064.769,A -85,B 0,C 180,E1 23299.201,E2 23299.201} C_VEL
LIN {X 0,Y 480.779,Z 1058.388,A -85,B 0,C 180,E1 23296.53,E2 23296.53} C_VEL
LIN {X 0,Y 481.734,Z 1049.553,A -85,B 0,C 180,E1 23293.604,E2 23293.604} C_VEL
LIN {X 0,Y 482.981,Z 1040.525,A -85,B 0,C 180,E1 23291.104,E2 23291.104} C_VEL
LIN {X 0,Y 484.994,Z 1028.127,A -85,B 0,C 180,E1 23288.217,E2 23288.217} C_VEL
LIN {X 0,Y 487.133,Z 1016.462,A -85,B 0,C 180,E1 23285.891,E2 23285.891} C_VEL
LIN {X 0,Y 490.255,Z 1000.843,A -85,B 0,C 180,E1 23283.209,E2 23283.209} C_VEL
LIN {X 0,Y 493.157,Z 986.966,A -85,B 0,C 180,E1 23281.148,E2 23281.148} C_VEL
LIN {X 0,Y 496.98,Z 969.373,A -85,B 0,C 180,E1 23278.864,E2 23278.864} C_VEL
LIN {X 0,Y 500.64,Z 952.33,A -85,B 0,C 180,E1 23276.959,E2 23276.959} C_VEL
LIN {X 0,Y 504.753,Z 933.076,A -85,B 0,C 180,E1 23275.076,E2 23275.076} C_VEL
LIN {X 0,Y 508.709,Z 913.527,A -85,B 0,C 180,E1 23273.447,E2 23273.447} C_VEL
LIN {X 0,Y 512.731,Z 892.926,A -85,B 0,C 180,E1 23271.958,E2 23271.958} C_VEL
LIN {X 0,Y 516.511,Z 871.435,A -85,B 0,C 180,E1 23270.655,E2 23270.655} C_VEL
LIN {X 0,Y 519.735,Z 851.531,A -85,B 0,C 180,E1 23269.627,E2 23269.627} C_VEL
LIN {X 0,Y 523.141,Z 827.416,A -85,B 0,C 180,E1 23268.6,E2 23268.6} C_VEL
LIN {X 0,Y 525.598,Z 807.062,A -85,B 0,C 180,E1 23267.904,E2 23267.904} C_VEL
LIN {X 0,Y 527.992,Z 783.427,A -85,B 0,C 180,E1 23267.264,E2 23267.264} C_VEL
LIN {X 0,Y 529.62,Z 758.915,A -85,B 0,C 180,E1 23266.792,E2 23266.792} C_VEL
LIN {X 0,Y 538.1,Z 522.434,A -85,B 0,C 180,E1 23263.314,E2 23263.314} C_VEL
LIN {X 0,Y 540.511,Z 453.255,A -85,B 0,C 180,E1 23262.278,E2 23262.278} C_VEL
LIN {X 0,Y 528.792,Z 432.769,A -85,B 0,C 180,E1 23260.506,E2 23260.506} C_VEL
LIN {X 0,Y 515.955,Z 412.163,A -85,B 0,C 180,E1 23258.433,E2 23258.433} C_VEL
LIN {X 0,Y 504.122,Z 394.665,A -85,B 0,C 180,E1 23256.374,E2 23256.374} C_VEL
LIN {X 0,Y 493.941,Z 380.422,A -85,B 0,C 180,E1 23254.458,E2 23254.458} C_VEL
LIN {X 0,Y 489.755,Z 374.884,A -85,B 0,C 180,E1 23253.627,E2 23253.627} C_VEL
LIN {X 0,Y 485.508,Z 369.065,A -85,B 0,C 180,E1 23252.725,E2 23252.725} C_VEL
LIN {X 0,Y 483.704,Z 365.21,A -85,B 0,C 180,E1 23251.812,E2 23251.812} C_VEL
LIN {X 0,Y 482.252,Z 362.279,A -85,B 0,C 180,E1 23251.083,E2 23251.083} C_VEL
LIN {X 0,Y 482.057,Z 361.159,A -85,B 0,C 180,E1 23250.819,E2 23250.819} C_VEL
LIN {X 0,Y 482.002,Z 361.162,A -85,B 0,C 180,E1 23247.394,E2 23247.394} C_VEL
LIN {X 0,Y 481.992,Z 361.164,A -85,B 0,C 180,E1 23243.815,E2 23243.815} C_VEL
LIN {X 0,Y 482.029,Z 361.175,A -85,B 0,C 180,E1 23240.348,E2 23240.348} C_VEL
LIN {X 0,Y 482.042,Z 361.186,A -85,B 0,C 180,E1 23236.758,E2 23236.758} C_VEL
LIN {X 0,Y 481.996,Z 361.17,A -85,B 0,C 180,E1 23233.313,E2 23233.313} C_VEL
LIN {X 0,Y 481.994,Z 361.158,A -85,B 0,C 180,E1 23229.674,E2 23229.674} C_VEL
LIN {X 0,Y 482.038,Z 361.178,A -85,B 0,C 180,E1 23226.192,E2 23226.192} C_VEL
LIN {X 0,Y 482.031,Z 361.179,A -85,B 0,C 180,E1 23222.616,E2 23222.616} C_VEL
LIN {X 0,Y 481.991,Z 361.155,A -85,B 0,C 180,E1 23219.168,E2 23219.168} C_VEL
LIN {X 0,Y 482.005,Z 361.18,A -85,B 0,C 180,E1 23215.598,E2 23215.598} C_VEL
LIN {X 0,Y 482.055,Z 361.176,A -85,B 0,C 180,E1 23212.132,E2 23212.132} C_VEL
LIN {X 0,Y 482.018,Z 361.154,A -85,B 0,C 180,E1 23208.513,E2 23208.513} C_VEL
LIN {X 0,Y 481.995,Z 361.175,A -85,B 0,C 180,E1 23205.094,E2 23205.094} C_VEL
LIN {X 0,Y 482.028,Z 361.188,A -85,B 0,C 180,E1 23201.621,E2 23201.621} C_VEL
LIN {X 0,Y 482.055,Z 361.164,A -85,B 0,C 180,E1 23197.999,E2 23197.999} C_VEL
LIN {X 0,Y 482.009,Z 361.16,A -85,B 0,C 180,E1 23194.438,E2 23194.438} C_VEL
LIN {X 0,Y 482,Z 361.166,A -85,B 0,C 180,E1 23190.96,E2 23190.96} C_VEL
LIN {X 0,Y 482.038,Z 361.169,A -85,B 0,C 180,E1 23187.504,E2 23187.504} C_VEL
LIN {X 0,Y 482.072,Z 361.362,A -85,B 0,C 180,E1 23185.655,E2 23185.655} C_VEL
LIN {X 0,Y 483.137,Z 364.357,A -85,B 0,C 180,E1 23185.382,E2 23185.382} C_VEL
LIN {X 0,Y 485.642,Z 366.951,A -85,B 0,C 180,E1 23184.868,E2 23184.868} C_VEL
LIN {X 0,Y 486.744,Z 367.867,A -85,B 0,C 180,E1 23184.651,E2 23184.651} C_VEL
LIN {X 0,Y 489.116,Z 371.544,A -85,B 0,C 180,E1 23184.148,E2 23184.148} C_VEL
LIN {X 0,Y 491.447,Z 373.923,A -85,B 0,C 180,E1 23183.696,E2 23183.696} C_VEL
LIN {X 0,Y 494.642,Z 378.163,A -85,B 0,C 180,E1 23183.067,E2 23183.067} C_VEL
LIN {X 0,Y 496.343,Z 380.199,A -85,B 0,C 180,E1 23182.745,E2 23182.745} C_VEL
LIN {X 0,Y 501.344,Z 386.76,A -85,B 0,C 180,E1 23181.81,E2 23181.81} C_VEL
LIN {X 0,Y 505.654,Z 392.322,A -85,B 0,C 180,E1 23181.037,E2 23181.037} C_VEL
LIN {X 0,Y 515.74,Z 405.857,A -85,B 0,C 180,E1 23179.314,E2 23179.314} C_VEL
LIN {X 0,Y 527.75,Z 423.031,A -85,B 0,C 180,E1 23177.401,E2 23177.401} C_VEL
LIN {X 0,Y 539.534,Z 442.323,A -85,B 0,C 180,E1 23175.623,E2 23175.623} C_VEL
LIN {X 0,Y 540.795,Z 444.867,A -85,B 0,C 180,E1 23175.432,E2 23175.432} C_VEL
LIN {X 0,Y 531.78,Z 692.251,A -85,B 0,C 180,E1 23171.804,E2 23171.804} C_VEL
LIN {X 0,Y 529.701,Z 745.554,A -85,B 0,C 180,E1 23170.997,E2 23170.997} C_VEL
LIN {X 0,Y 527.831,Z 769.887,A -85,B 0,C 180,E1 23170.452,E2 23170.452} C_VEL
LIN {X 0,Y 525.596,Z 792.386,A -85,B 0,C 180,E1 23169.787,E2 23169.787} C_VEL
LIN {X 0,Y 522.608,Z 816.404,A -85,B 0,C 180,E1 23168.87,E2 23168.87} C_VEL
LIN {X 0,Y 519.646,Z 836.867,A -85,B 0,C 180,E1 23167.916,E2 23167.916} C_VEL
LIN {X 0,Y 515.736,Z 860.378,A -85,B 0,C 180,E1 23166.596,E2 23166.596} C_VEL
LIN {X 0,Y 512.213,Z 879.579,A -85,B 0,C 180,E1 23165.315,E2 23165.315} C_VEL
LIN {X 0,Y 507.952,Z 900.99,A -85,B 0,C 180,E1 23163.65,E2 23163.65} C_VEL
LIN {X 0,Y 504.181,Z 918.716,A -85,B 0,C 180,E1 23162.04,E2 23162.04} C_VEL
LIN {X 0,Y 500.171,Z 937.19,A -85,B 0,C 180,E1 23160.117,E2 23160.117} C_VEL
LIN {X 0,Y 498.41,Z 944.959,A -85,B 0,C 180,E1 23159.204,E2 23159.204} C_VEL
LIN {X 0,Y 496.317,Z 950.385,A -85,B 0,C 180,E1 23158.607,E2 23158.607} C_VEL
LIN {X 0,Y 487.897,Z 963.83,A -85,B 0,C 180,E1 23157.163,E2 23157.163} C_VEL
LIN {X 0,Y 485.877,Z 968.773,A -85,B 0,C 180,E1 23156.505,E2 23156.505} C_VEL
LIN {X 0,Y 482.467,Z 983.638,A -85,B 0,C 180,E1 23154.096,E2 23154.096} C_VEL
LIN {X 0,Y 479.877,Z 995.452,A -85,B 0,C 180,E1 23151.899,E2 23151.899} C_VEL
LIN {X 0,Y 477.214,Z 1008.531,A -85,B 0,C 180,E1 23149.078,E2 23149.078} C_VEL
LIN {X 0,Y 475.439,Z 1018.17,A -85,B 0,C 180,E1 23146.62,E2 23146.62} C_VEL
LIN {X 0,Y 473.969,Z 1027.637,A -85,B 0,C 180,E1 23143.791,E2 23143.791} C_VEL
LIN {X 0,Y 472.98,Z 1035.212,A -85,B 0,C 180,E1 23140.968,E2 23140.968} C_VEL
LIN {X 0,Y 472.403,Z 1041.087,A -85,B 0,C 180,E1 23138.275,E2 23138.275} C_VEL
LIN {X 0,Y 472.095,Z 1045.818,A -85,B 0,C 180,E1 23135.347,E2 23135.347} C_VEL
LIN {X 0,Y 471.981,Z 1048.666,A -85,B 0,C 180,E1 23132.793,E2 23132.793} C_VEL
LIN {X 0,Y 471.951,Z 1050.529,A -85,B 0,C 180,E1 23129.964,E2 23129.964} C_VEL
LIN {X 0,Y 471.933,Z 1050.767,A -85,B 0,C 180,E1 23127.085,E2 23127.085} C_VEL
LIN {X 0,Y 471.954,Z 1049.871,A -85,B 0,C 180,E1 23124.651,E2 23124.651} C_VEL
LIN {X 0,Y 472.044,Z 1047.586,A -85,B 0,C 180,E1 23121.841,E2 23121.841} C_VEL
LIN {X 0,Y 472.23,Z 1043.669,A -85,B 0,C 180,E1 23119.014,E2 23119.014} C_VEL
LIN {X 0,Y 472.641,Z 1038.856,A -85,B 0,C 180,E1 23116.419,E2 23116.419} C_VEL
LIN {X 0,Y 473.523,Z 1031.375,A -85,B 0,C 180,E1 23113.311,E2 23113.311} C_VEL
LIN {X 0,Y 474.623,Z 1023.93,A -85,B 0,C 180,E1 23110.813,E2 23110.813} C_VEL
LIN {X 0,Y 476.439,Z 1013.732,A -85,B 0,C 180,E1 23107.935,E2 23107.935} C_VEL
LIN {X 0,Y 478.686,Z 1002.549,A -85,B 0,C 180,E1 23105.306,E2 23105.306} C_VEL
LIN {X 0,Y 481.571,Z 989.664,A -85,B 0,C 180,E1 23102.686,E2 23102.686} C_VEL
LIN {X 0,Y 484.842,Z 975.551,A -85,B 0,C 180,E1 23100.254,E2 23100.254} C_VEL
LIN {X 0,Y 488.67,Z 959.912,A -85,B 0,C 180,E1 23097.899,E2 23097.899} C_VEL
LIN {X 0,Y 492.747,Z 942.996,A -85,B 0,C 180,E1 23095.729,E2 23095.729} C_VEL
LIN {X 0,Y 497.039,Z 925.273,A -85,B 0,C 180,E1 23093.741,E2 23093.741} C_VEL
LIN {X 0,Y 501.465,Z 905.971,A -85,B 0,C 180,E1 23091.897,E2 23091.897} C_VEL
LIN {X 0,Y 505.714,Z 886.807,A -85,B 0,C 180,E1 23090.31,E2 23090.31} C_VEL
LIN {X 0,Y 510.061,Z 865.297,A -85,B 0,C 180,E1 23088.801,E2 23088.801} C_VEL
LIN {X 0,Y 513.423,Z 847.177,A -85,B 0,C 180,E1 23087.712,E2 23087.712} C_VEL
LIN {X 0,Y 517.343,Z 823.726,A -85,B 0,C 180,E1 23086.524,E2 23086.524} C_VEL
LIN {X 0,Y 520.212,Z 803.366,A -85,B 0,C 180,E1 23085.679,E2 23085.679} C_VEL
LIN {X 0,Y 522.826,Z 781.873,A -85,B 0,C 180,E1 23084.949,E2 23084.949} C_VEL
LIN {X 0,Y 525.117,Z 757.355,A -85,B 0,C 180,E1 23084.316,E2 23084.316} C_VEL
LIN {X 0,Y 526.51,Z 735.76,A -85,B 0,C 180,E1 23083.907,E2 23083.907} C_VEL
LIN {X 0,Y 536.423,Z 486.99,A -85,B 0,C 180,E1 23080.207,E2 23080.207} C_VEL
LIN {X 0,Y 537.887,Z 449.193,A -85,B 0,C 180,E1 23079.631,E2 23079.631} C_VEL
LIN {X 0,Y 526.627,Z 430.909,A -85,B 0,C 180,E1 23077.792,E2 23077.792} C_VEL
LIN {X 0,Y 515.323,Z 415.027,A -85,B 0,C 180,E1 23075.838,E2 23075.838} C_VEL
LIN {X 0,Y 505.137,Z 401.359,A -85,B 0,C 180,E1 23073.932,E2 23073.932} C_VEL
LIN {X 0,Y 497.21,Z 391.268,A -85,B 0,C 180,E1 23072.339,E2 23072.339} C_VEL
LIN {X 0,Y 492.535,Z 385.487,A -85,B 0,C 180,E1 23071.347,E2 23071.347} C_VEL
LIN {X 0,Y 489.056,Z 380.901,A -85,B 0,C 180,E1 23070.569,E2 23070.569} C_VEL
LIN {X 0,Y 485.457,Z 377.109,A -85,B 0,C 180,E1 23069.761,E2 23069.761} C_VEL
LIN {X 0,Y 483.938,Z 374.706,A -85,B 0,C 180,E1 23069.388,E2 23069.388} C_VEL
LIN {X 0,Y 480.759,Z 371.783,A -85,B 0,C 180,E1 23068.646,E2 23068.646} C_VEL
LIN {X 0,Y 478.908,Z 368.519,A -85,B 0,C 180,E1 23068.155,E2 23068.155} C_VEL
LIN {X 0,Y 475.901,Z 366.357,A -85,B 0,C 180,E1 23067.43,E2 23067.43} C_VEL
LIN {X 0,Y 474.353,Z 363.538,A -85,B 0,C 180,E1 23066.992,E2 23066.992} C_VEL
LIN {X 0,Y 474.067,Z 362.181,A -85,B 0,C 180,E1 23066.852,E2 23066.852} C_VEL
LIN {X 0,Y 474.061,Z 362.181,A -85,B 0,C 180,E1 23063.23,E2 23063.23} C_VEL
LIN {X 0,Y 474.095,Z 362.177,A -85,B 0,C 180,E1 23059.722,E2 23059.722} C_VEL
LIN {X 0,Y 474.101,Z 362.174,A -85,B 0,C 180,E1 23056.164,E2 23056.164} C_VEL
LIN {X 0,Y 474.06,Z 362.171,A -85,B 0,C 180,E1 23052.671,E2 23052.671} C_VEL
LIN {X 0,Y 474.056,Z 362.163,A -85,B 0,C 180,E1 23048.98,E2 23048.98} C_VEL
LIN {X 0,Y 474.095,Z 362.151,A -85,B 0,C 180,E1 23045.567,E2 23045.567} C_VEL
LIN {X 0,Y 474.085,Z 362.155,A -85,B 0,C 180,E1 23042.055,E2 23042.055} C_VEL
LIN {X 0,Y 474.057,Z 362.173,A -85,B 0,C 180,E1 23038.55,E2 23038.55} C_VEL
LIN {X 0,Y 474.063,Z 362.18,A -85,B 0,C 180,E1 23034.918,E2 23034.918} C_VEL
LIN {X 0,Y 474.103,Z 362.165,A -85,B 0,C 180,E1 23031.388,E2 23031.388} C_VEL
LIN {X 0,Y 474.084,Z 362.154,A -85,B 0,C 180,E1 23027.824,E2 23027.824} C_VEL
LIN {X 0,Y 474.053,Z 362.153,A -85,B 0,C 180,E1 23024.337,E2 23024.337} C_VEL
LIN {X 0,Y 474.065,Z 362.152,A -85,B 0,C 180,E1 23020.79,E2 23020.79} C_VEL
LIN {X 0,Y 474.119,Z 362.15,A -85,B 0,C 180,E1 23017.298,E2 23017.298} C_VEL
LIN {X 0,Y 474.078,Z 362.158,A -85,B 0,C 180,E1 23013.686,E2 23013.686} C_VEL
LIN {X 0,Y 474.077,Z 362.315,A -85,B 0,C 180,E1 23012.354,E2 23012.354} C_VEL
LIN {X 0,Y 475.302,Z 365.501,A -85,B 0,C 180,E1 23011.475,E2 23011.475} C_VEL
LIN {X 0,Y 476.519,Z 367.356,A -85,B 0,C 180,E1 23010.869,E2 23010.869} C_VEL
LIN {X 0,Y 477.305,Z 369.143,A -85,B 0,C 180,E1 23010.508,E2 23010.508} C_VEL
LIN {X 0,Y 481.628,Z 374.484,A -85,B 0,C 180,E1 23009.427,E2 23009.427} C_VEL
LIN {X 0,Y 485.846,Z 379.99,A -85,B 0,C 180,E1 23008.414,E2 23008.414} C_VEL
LIN {X 0,Y 489.056,Z 383.993,A -85,B 0,C 180,E1 23007.68,E2 23007.68} C_VEL
LIN {X 0,Y 496.592,Z 394.098,A -85,B 0,C 180,E1 23006.031,E2 23006.031} C_VEL
LIN {X 0,Y 508.11,Z 410.227,A -85,B 0,C 180,E1 23003.712,E2 23003.712} C_VEL
LIN {X 0,Y 520.51,Z 429.063,A -85,B 0,C 180,E1 23001.429,E2 23001.429} C_VEL
LIN {X 0,Y 532.363,Z 448.497,A -85,B 0,C 180,E1 22999.416,E2 22999.416} C_VEL
LIN {X 0,Y 537.829,Z 458.36,A -85,B 0,C 180,E1 22998.526,E2 22998.526} C_VEL
LIN {X 0,Y 527.95,Z 707.107,A -85,B 0,C 180,E1 22994.83,E2 22994.83} C_VEL
LIN {X 0,Y 525.528,Z 765.296,A -85,B 0,C 180,E1 22993.942,E2 22993.942} C_VEL
LIN {X 0,Y 523.396,Z 790.049,A -85,B 0,C 180,E1 22993.404,E2 22993.404} C_VEL
LIN {X 0,Y 521.086,Z 810.719,A -85,B 0,C 180,E1 22992.813,E2 22992.813} C_VEL
LIN {X 0,Y 517.774,Z 835.01,A -85,B 0,C 180,E1 22991.926,E2 22991.926} C_VEL
LIN {X 0,Y 514.5,Z 855.632,A -85,B 0,C 180,E1 22990.988,E2 22990.988} C_VEL
LIN {X 0,Y 510.642,Z 877.43,A -85,B 0,C 180,E1 22989.814,E2 22989.814} C_VEL
LIN {X 0,Y 506.471,Z 898.347,A -85,B 0,C 180,E1 22988.454,E2 22988.454} C_VEL
LIN {X 0,Y 502.284,Z 918.212,A -85,B 0,C 180,E1 22986.955,E2 22986.955} C_VEL
LIN {X 0,Y 497.705,Z 938.553,A -85,B 0,C 180,E1 22985.148,E2 22985.148} C_VEL
LIN {X 0,Y 493.798,Z 955.453,A -85,B 0,C 180,E1 22983.42,E2 22983.42} C_VEL
LIN {X 0,Y 489.242,Z 974.735,A -85,B 0,C 180,E1 22981.136,E2 22981.136} C_VEL
LIN {X 0,Y 485.715,Z 989.848,A -85,B 0,C 180,E1 22979.067,E2 22979.067} C_VEL
LIN {X 0,Y 482.023,Z 1006.171,A -85,B 0,C 180,E1 22976.487,E2 22976.487} C_VEL
LIN {X 0,Y 479.406,Z 1018.351,A -85,B 0,C 180,E1 22974.26,E2 22974.26} C_VEL
LIN {X 0,Y 476.858,Z 1031.376,A -85,B 0,C 180,E1 22971.527,E2 22971.527} C_VEL
LIN {X 0,Y 475.034,Z 1041.882,A -85,B 0,C 180,E1 22968.914,E2 22968.914} C_VEL
LIN {X 0,Y 473.667,Z 1051.389,A -85,B 0,C 180,E1 22966.16,E2 22966.16} C_VEL
LIN {X 0,Y 472.751,Z 1059.313,A -85,B 0,C 180,E1 22963.329,E2 22963.329} C_VEL
LIN {X 0,Y 472.269,Z 1065.163,A -85,B 0,C 180,E1 22960.769,E2 22960.769} C_VEL
LIN {X 0,Y 471.994,Z 1070.392,A -85,B 0,C 180,E1 22957.792,E2 22957.792} C_VEL
LIN {X 0,Y 471.942,Z 1073.478,A -85,B 0,C 180,E1 22955.227,E2 22955.227} C_VEL
LIN {X 0,Y 471.932,Z 1075.375,A -85,B 0,C 180,E1 22952.672,E2 22952.672} C_VEL
LIN {X 0,Y 471.932,Z 1076.059,A -85,B 0,C 180,E1 22949.757,E2 22949.757} C_VEL
LIN {X 0,Y 471.934,Z 1075.268,A -85,B 0,C 180,E1 22947.207,E2 22947.207} C_VEL
LIN {X 0,Y 471.944,Z 1073.375,A -85,B 0,C 180,E1 22944.733,E2 22944.733} C_VEL
LIN {X 0,Y 472.022,Z 1069.754,A -85,B 0,C 180,E1 22941.841,E2 22941.841} C_VEL
LIN {X 0,Y 472.281,Z 1064.788,A -85,B 0,C 180,E1 22939.139,E2 22939.139} C_VEL
LIN {X 0,Y 472.774,Z 1058.76,A -85,B 0,C 180,E1 22936.547,E2 22936.547} C_VEL
LIN {X 0,Y 473.804,Z 1049.706,A -85,B 0,C 180,E1 22933.447,E2 22933.447} C_VEL
LIN {X 0,Y 475.071,Z 1040.927,A -85,B 0,C 180,E1 22930.96,E2 22930.96} C_VEL
LIN {X 0,Y 477.104,Z 1029.013,A -85,B 0,C 180,E1 22928.097,E2 22928.097} C_VEL
LIN {X 0,Y 479.435,Z 1016.819,A -85,B 0,C 180,E1 22925.61,E2 22925.61} C_VEL
LIN {X 0,Y 482.539,Z 1002.044,A -85,B 0,C 180,E1 22923.003,E2 22923.003} C_VEL
LIN {X 0,Y 485.708,Z 987.476,A -85,B 0,C 180,E1 22920.793,E2 22920.793} C_VEL
LIN {X 0,Y 489.566,Z 970.579,A -85,B 0,C 180,E1 22918.545,E2 22918.545} C_VEL
LIN {X 0,Y 493.463,Z 953.107,A -85,B 0,C 180,E1 22916.554,E2 22916.554} C_VEL
LIN {X 0,Y 497.58,Z 934.629,A -85,B 0,C 180,E1 22914.709,E2 22914.709} C_VEL
LIN {X 0,Y 501.813,Z 914.624,A -85,B 0,C 180,E1 22913.005,E2 22913.005} C_VEL
LIN {X 0,Y 505.617,Z 895.798,A -85,B 0,C 180,E1 22911.614,E2 22911.614} C_VEL
LIN {X 0,Y 509.903,Z 872.784,A -85,B 0,C 180,E1 22910.173,E2 22910.173} C_VEL
LIN {X 0,Y 513.29,Z 852.643,A -85,B 0,C 180,E1 22909.116,E2 22909.116} C_VEL
LIN {X 0,Y 516.792,Z 829.09,A -85,B 0,C 180,E1 22908.088,E2 22908.088} C_VEL
LIN {X 0,Y 519.471,Z 807.679,A -85,B 0,C 180,E1 22907.344,E2 22907.344} C_VEL
LIN {X 0,Y 521.775,Z 785.818,A -85,B 0,C 180,E1 22906.74,E2 22906.74} C_VEL
LIN {X 0,Y 523.623,Z 760.497,A -85,B 0,C 180,E1 22906.23,E2 22906.23} C_VEL
LIN {X 0,Y 532.18,Z 531.278,A -85,B 0,C 180,E1 22902.828,E2 22902.828} C_VEL
LIN {X 0,Y 534.969,Z 456.72,A -85,B 0,C 180,E1 22901.712,E2 22901.712} C_VEL
LIN {X 0,Y 522.845,Z 435.554,A -85,B 0,C 180,E1 22899.823,E2 22899.823} C_VEL
LIN {X 0,Y 511.086,Z 416.727,A -85,B 0,C 180,E1 22897.867,E2 22897.867} C_VEL
LIN {X 0,Y 500.477,Z 400.882,A -85,B 0,C 180,E1 22895.971,E2 22895.971} C_VEL
LIN {X 0,Y 490.284,Z 386.534,A -85,B 0,C 180,E1 22894.008,E2 22894.008} C_VEL
LIN {X 0,Y 486.274,Z 381.192,A -85,B 0,C 180,E1 22893.194,E2 22893.194} C_VEL
LIN {X 0,Y 481.995,Z 375.418,A -85,B 0,C 180,E1 22892.288,E2 22892.288} C_VEL
LIN {X 0,Y 476.729,Z 368.369,A -85,B 0,C 180,E1 22891.062,E2 22891.062} C_VEL
LIN {X 0,Y 475.888,Z 366.287,A -85,B 0,C 180,E1 22890.562,E2 22890.562} C_VEL
LIN {X 0,Y 474.21,Z 363.024,A -85,B 0,C 180,E1 22889.69,E2 22889.69} C_VEL
LIN {X 0,Y 474.064,Z 362.171,A -85,B 0,C 180,E1 22889.505,E2 22889.505} C_VEL
LIN {X 0,Y 474.057,Z 362.168,A -85,B 0,C 180,E1 22885.888,E2 22885.888} C_VEL
LIN {X 0,Y 474.081,Z 362.155,A -85,B 0,C 180,E1 22882.312,E2 22882.312} C_VEL
LIN {X 0,Y 474.102,Z 362.144,A -85,B 0,C 180,E1 22878.747,E2 22878.747} C_VEL
LIN {X 0,Y 474.061,Z 362.157,A -85,B 0,C 180,E1 22875.287,E2 22875.287} C_VEL
LIN {X 0,Y 474.06,Z 362.179,A -85,B 0,C 180,E1 22871.682,E2 22871.682} C_VEL
LIN {X 0,Y 474.087,Z 362.157,A -85,B 0,C 180,E1 22868.124,E2 22868.124} C_VEL
LIN {X 0,Y 474.083,Z 362.143,A -85,B 0,C 180,E1 22864.718,E2 22864.718} C_VEL
LIN {X 0,Y 474.058,Z 362.177,A -85,B 0,C 180,E1 22861.209,E2 22861.209} C_VEL
LIN {X 0,Y 474.062,Z 362.164,A -85,B 0,C 180,E1 22857.582,E2 22857.582} C_VEL
LIN {X 0,Y 474.104,Z 362.14,A -85,B 0,C 180,E1 22854.068,E2 22854.068} C_VEL
LIN {X 0,Y 474.074,Z 362.171,A -85,B 0,C 180,E1 22850.653,E2 22850.653} C_VEL
LIN {X 0,Y 474.059,Z 362.17,A -85,B 0,C 180,E1 22847.081,E2 22847.081} C_VEL
LIN {X 0,Y 474.078,Z 362.146,A -85,B 0,C 180,E1 22843.583,E2 22843.583} C_VEL
LIN {X 0,Y 474.111,Z 362.15,A -85,B 0,C 180,E1 22840.022,E2 22840.022} C_VEL
LIN {X 0,Y 474.072,Z 362.179,A -85,B 0,C 180,E1 22836.507,E2 22836.507} C_VEL
LIN {X 0,Y 474.063,Z 362.176,A -85,B 0,C 180,E1 22832.883,E2 22832.883} C_VEL
LIN {X 0,Y 474.078,Z 362.162,A -85,B 0,C 180,E1 22829.309,E2 22829.309} C_VEL
LIN {X 0,Y 474.091,Z 362.308,A -85,B 0,C 180,E1 22827.142,E2 22827.142} C_VEL
LIN {X 0,Y 475.104,Z 365.228,A -85,B 0,C 180,E1 22826.861,E2 22826.861} C_VEL
LIN {X 0,Y 477.626,Z 367.858,A -85,B 0,C 180,E1 22826.305,E2 22826.305} C_VEL
LIN {X 0,Y 478.935,Z 368.872,A -85,B 0,C 180,E1 22826.032,E2 22826.032} C_VEL
LIN {X 0,Y 481.212,Z 372.548,A -85,B 0,C 180,E1 22825.513,E2 22825.513} C_VEL
LIN {X 0,Y 483.785,Z 375.045,A -85,B 0,C 180,E1 22824.984,E2 22824.984} C_VEL
LIN {X 0,Y 486.936,Z 379.219,A -85,B 0,C 180,E1 22824.326,E2 22824.326} C_VEL
LIN {X 0,Y 488.583,Z 381.187,A -85,B 0,C 180,E1 22823.994,E2 22823.994} C_VEL
LIN {X 0,Y 492.304,Z 385.682,A -85,B 0,C 180,E1 22823.263,E2 22823.263} C_VEL
LIN {X 0,Y 504.843,Z 402.265,A -85,B 0,C 180,E1 22820.929,E2 22820.929} C_VEL
LIN {X 0,Y 517.409,Z 419.65,A -85,B 0,C 180,E1 22818.796,E2 22818.796} C_VEL
LIN {X 0,Y 527.401,Z 434.855,A -85,B 0,C 180,E1 22817.206,E2 22817.206} C_VEL
LIN {X 0,Y 535.203,Z 448.273,A -85,B 0,C 180,E1 22816.007,E2 22816.007} C_VEL
LIN {X 0,Y 525.824,Z 696.07,A -85,B 0,C 180,E1 22812.346,E2 22812.346} C_VEL
LIN {X 0,Y 523.772,Z 746.313,A -85,B 0,C 180,E1 22811.575,E2 22811.575} C_VEL
LIN {X 0,Y 521.832,Z 770.517,A -85,B 0,C 180,E1 22811.026,E2 22811.026} C_VEL
LIN {X 0,Y 519.46,Z 793.618,A -85,B 0,C 180,E1 22810.335,E2 22810.335} C_VEL
LIN {X 0,Y 516.413,Z 817.049,A -85,B 0,C 180,E1 22809.426,E2 22809.426} C_VEL
LIN {X 0,Y 513.235,Z 838.261,A -85,B 0,C 180,E1 22808.424,E2 22808.424} C_VEL
LIN {X 0,Y 509.311,Z 860.899,A -85,B 0,C 180,E1 22807.135,E2 22807.135} C_VEL
LIN {X 0,Y 505.778,Z 879.483,A -85,B 0,C 180,E1 22805.885,E2 22805.885} C_VEL
LIN {X 0,Y 501.402,Z 900.777,A -85,B 0,C 180,E1 22804.219,E2 22804.219} C_VEL
LIN {X 0,Y 497.476,Z 918.544,A -85,B 0,C 180,E1 22802.592,E2 22802.592} C_VEL
LIN {X 0,Y 493.285,Z 937.085,A -85,B 0,C 180,E1 22800.65,E2 22800.65} C_VEL
LIN {X 0,Y 489.304,Z 954.023,A -85,B 0,C 180,E1 22798.566,E2 22798.566} C_VEL
LIN {X 0,Y 485.877,Z 968.773,A -85,B 0,C 180,E1 22796.505,E2 22796.505} C_VEL
LIN {X 0,Y 483.874,Z 973.63,A -85,B 0,C 180,E1 22795.829,E2 22795.829} C_VEL
LIN {X 0,Y 475.222,Z 986.194,A -85,B 0,C 180,E1 22794.061,E2 22794.061} C_VEL
LIN {X 0,Y 473.68,Z 989.946,A -85,B 0,C 180,E1 22793.424,E2 22793.424} C_VEL
LIN {X 0,Y 470.77,Z 1002.847,A -85,B 0,C 180,E1 22790.775,E2 22790.775} C_VEL
LIN {X 0,Y 468.526,Z 1013.891,A -85,B 0,C 180,E1 22788.155,E2 22788.155} C_VEL
LIN {X 0,Y 466.697,Z 1023.986,A -85,B 0,C 180,E1 22785.279,E2 22785.279} C_VEL
LIN {X 0,Y 465.534,Z 1031.723,A -85,B 0,C 180,E1 22782.655,E2 22782.655} C_VEL
LIN {X 0,Y 464.646,Z 1039.108,A -85,B 0,C 180,E1 22779.538,E2 22779.538} C_VEL
LIN {X 0,Y 464.235,Z 1043.881,A -85,B 0,C 180,E1 22776.928,E2 22776.928} C_VEL
LIN {X 0,Y 464.026,Z 1047.9,A -85,B 0,C 180,E1 22773.954,E2 22773.954} C_VEL
LIN {X 0,Y 463.956,Z 1050.135,A -85,B 0,C 180,E1 22771.111,E2 22771.111} C_VEL
LIN {X 0,Y 463.931,Z 1050.997,A -85,B 0,C 180,E1 22768.641,E2 22768.641} C_VEL
LIN {X 0,Y 463.948,Z 1050.673,A -85,B 0,C 180,E1 22765.674,E2 22765.674} C_VEL
LIN {X 0,Y 463.995,Z 1048.902,A -85,B 0,C 180,E1 22762.944,E2 22762.944} C_VEL
LIN {X 0,Y 464.117,Z 1046.206,A -85,B 0,C 180,E1 22760.451,E2 22760.451} C_VEL
LIN {X 0,Y 464.468,Z 1041.533,A -85,B 0,C 180,E1 22757.442,E2 22757.442} C_VEL
LIN {X 0,Y 465.106,Z 1035.651,A -85,B 0,C 180,E1 22754.667,E2 22754.667} C_VEL
LIN {X 0,Y 466.216,Z 1028.038,A -85,B 0,C 180,E1 22751.752,E2 22751.752} C_VEL
LIN {X 0,Y 467.861,Z 1018.5,A -85,B 0,C 180,E1 22748.827,E2 22748.827} C_VEL
LIN {X 0,Y 469.943,Z 1008.241,A -85,B 0,C 180,E1 22746.155,E2 22746.155} C_VEL
LIN {X 0,Y 472.807,Z 995.484,A -85,B 0,C 180,E1 22743.363,E2 22743.363} C_VEL
LIN {X 0,Y 475.941,Z 982.559,A -85,B 0,C 180,E1 22740.923,E2 22740.923} C_VEL
LIN {X 0,Y 479.752,Z 967.335,A -85,B 0,C 180,E1 22738.458,E2 22738.458} C_VEL
LIN {X 0,Y 483.558,Z 952.326,A -85,B 0,C 180,E1 22736.347,E2 22736.347} C_VEL
LIN {X 0,Y 488.246,Z 933.889,A -85,B 0,C 180,E1 22734.11,E2 22734.11} C_VEL
LIN {X 0,Y 492.302,Z 917.405,A -85,B 0,C 180,E1 22732.383,E2 22732.383} C_VEL
LIN {X 0,Y 496.988,Z 897.686,A -85,B 0,C 180,E1 22730.586,E2 22730.586} C_VEL
LIN {X 0,Y 501.299,Z 877.962,A -85,B 0,C 180,E1 22729.06,E2 22729.06} C_VEL
LIN {X 0,Y 505.556,Z 857.141,A -85,B 0,C 180,E1 22727.672,E2 22727.672} C_VEL
LIN {X 0,Y 509.508,Z 835.23,A -85,B 0,C 180,E1 22726.463,E2 22726.463} C_VEL
LIN {X 0,Y 512.898,Z 813.975,A -85,B 0,C 180,E1 22725.475,E2 22725.475} C_VEL
LIN {X 0,Y 516.16,Z 789.465,A -85,B 0,C 180,E1 22724.565,E2 22724.565} C_VEL
LIN {X 0,Y 518.534,Z 767.49,A -85,B 0,C 180,E1 22723.927,E2 22723.927} C_VEL
LIN {X 0,Y 520.571,Z 741.414,A -85,B 0,C 180,E1 22723.377,E2 22723.377} C_VEL
LIN {X 0,Y 530.094,Z 511.949,A -85,B 0,C 180,E1 22719.927,E2 22719.927} C_VEL
LIN {X 0,Y 532.528,Z 452.842,A -85,B 0,C 180,E1 22719.029,E2 22719.029} C_VEL
LIN {X 0,Y 522.36,Z 436.353,A -85,B 0,C 180,E1 22717.324,E2 22717.324} C_VEL
LIN {X 0,Y 510.049,Z 418.773,A -85,B 0,C 180,E1 22715.126,E2 22715.126} C_VEL
LIN {X 0,Y 498.444,Z 403.366,A -85,B 0,C 180,E1 22712.863,E2 22712.863} C_VEL
LIN {X 0,Y 493.337,Z 397.077,A -85,B 0,C 180,E1 22711.801,E2 22711.801} C_VEL
LIN {X 0,Y 489.447,Z 392.132,A -85,B 0,C 180,E1 22710.951,E2 22710.951} C_VEL
LIN {X 0,Y 485.415,Z 387.125,A -85,B 0,C 180,E1 22710.036,E2 22710.036} C_VEL
LIN {X 0,Y 481.938,Z 382.81,A -85,B 0,C 180,E1 22709.215,E2 22709.215} C_VEL
LIN {X 0,Y 480.711,Z 381.436,A -85,B 0,C 180,E1 22708.921,E2 22708.921} C_VEL
LIN {X 0,Y 477.53,Z 377.878,A -85,B 0,C 180,E1 22708.141,E2 22708.141} C_VEL
LIN {X 0,Y 476.191,Z 375.752,A -85,B 0,C 180,E1 22707.785,E2 22707.785} C_VEL
LIN {X 0,Y 473.057,Z 372.975,A -85,B 0,C 180,E1 22706.995,E2 22706.995} C_VEL
LIN {X 0,Y 471.22,Z 369.639,A -85,B 0,C 180,E1 22706.462,E2 22706.462} C_VEL
LIN {X 0,Y 467.964,Z 367.324,A -85,B 0,C 180,E1 22705.604,E2 22705.604} C_VEL
LIN {X 0,Y 466.4,Z 364.474,A -85,B 0,C 180,E1 22705.118,E2 22705.118} C_VEL
LIN {X 0,Y 466.12,Z 363.148,A -85,B 0,C 180,E1 22704.998,E2 22704.998} C_VEL
LIN {X 0,Y 466.127,Z 363.146,A -85,B 0,C 180,E1 22701.387,E2 22701.387} C_VEL
LIN {X 0,Y 466.163,Z 363.141,A -85,B 0,C 180,E1 22697.862,E2 22697.862} C_VEL
LIN {X 0,Y 466.146,Z 363.143,A -85,B 0,C 180,E1 22694.281,E2 22694.281} C_VEL
LIN {X 0,Y 466.118,Z 363.151,A -85,B 0,C 180,E1 22690.742,E2 22690.742} C_VEL
LIN {X 0,Y 466.121,Z 363.16,A -85,B 0,C 180,E1 22687.023,E2 22687.023} C_VEL
LIN {X 0,Y 466.15,Z 363.166,A -85,B 0,C 180,E1 22683.443,E2 22683.443} C_VEL
LIN {X 0,Y 466.178,Z 363.156,A -85,B 0,C 180,E1 22679.754,E2 22679.754} C_VEL
LIN {X 0,Y 466.138,Z 363.149,A -85,B 0,C 180,E1 22676.064,E2 22676.064} C_VEL
LIN {X 0,Y 466.114,Z 363.143,A -85,B 0,C 180,E1 22672.481,E2 22672.481} C_VEL
LIN {X 0,Y 466.124,Z 363.141,A -85,B 0,C 180,E1 22668.868,E2 22668.868} C_VEL
LIN {X 0,Y 466.17,Z 363.14,A -85,B 0,C 180,E1 22665.319,E2 22665.319} C_VEL
LIN {X 0,Y 466.156,Z 363.147,A -85,B 0,C 180,E1 22661.62,E2 22661.62} C_VEL
LIN {X 0,Y 466.12,Z 363.16,A -85,B 0,C 180,E1 22658.083,E2 22658.083} C_VEL
LIN {X 0,Y 466.12,Z 363.164,A -85,B 0,C 180,E1 22654.458,E2 22654.458} C_VEL
LIN {X 0,Y 466.144,Z 363.338,A -85,B 0,C 180,E1 22654.05,E2 22654.05} C_VEL
LIN {X 0,Y 467.734,Z 367.014,A -85,B 0,C 180,E1 22652.913,E2 22652.913} C_VEL
LIN {X 0,Y 468.874,Z 368.515,A -85,B 0,C 180,E1 22652.469,E2 22652.469} C_VEL
LIN {X 0,Y 471.856,Z 372.619,A -85,B 0,C 180,E1 22651.628,E2 22651.628} C_VEL
LIN {X 0,Y 474.05,Z 375.053,A -85,B 0,C 180,E1 22651.048,E2 22651.048} C_VEL
LIN {X 0,Y 477.533,Z 379.466,A -85,B 0,C 180,E1 22650.144,E2 22650.144} C_VEL
LIN {X 0,Y 486.363,Z 391.096,A -85,B 0,C 180,E1 22648.001,E2 22648.001} C_VEL
LIN {X 0,Y 493.35,Z 400.497,A -85,B 0,C 180,E1 22646.441,E2 22646.441} C_VEL
LIN {X 0,Y 504.851,Z 416.811,A -85,B 0,C 180,E1 22644.074,E2 22644.074} C_VEL
LIN {X 0,Y 517.021,Z 435.55,A -85,B 0,C 180,E1 22641.784,E2 22641.784} C_VEL
LIN {X 0,Y 528.515,Z 454.634,A -85,B 0,C 180,E1 22639.789,E2 22639.789} C_VEL
LIN {X 0,Y 532.466,Z 461.98,A -85,B 0,C 180,E1 22639.125,E2 22639.125} C_VEL
LIN {X 0,Y 522.243,Z 710.056,A -85,B 0,C 180,E1 22635.414,E2 22635.414} C_VEL
LIN {X 0,Y 519.837,Z 765.471,A -85,B 0,C 180,E1 22634.559,E2 22634.559} C_VEL
LIN {X 0,Y 517.64,Z 790.07,A -85,B 0,C 180,E1 22634.02,E2 22634.02} C_VEL
LIN {X 0,Y 515.264,Z 810.646,A -85,B 0,C 180,E1 22633.428,E2 22633.428} C_VEL
LIN {X 0,Y 511.812,Z 835.1,A -85,B 0,C 180,E1 22632.528,E2 22632.528} C_VEL
LIN {X 0,Y 508.624,Z 854.555,A -85,B 0,C 180,E1 22631.641,E2 22631.641} C_VEL
LIN {X 0,Y 504.616,Z 876.537,A -85,B 0,C 180,E1 22630.457,E2 22630.457} C_VEL
LIN {X 0,Y 500.294,Z 897.508,A -85,B 0,C 180,E1 22629.091,E2 22629.091} C_VEL
LIN {X 0,Y 496.097,Z 916.695,A -85,B 0,C 180,E1 22627.64,E2 22627.64} C_VEL
LIN {X 0,Y 491.136,Z 937.933,A -85,B 0,C 180,E1 22625.753,E2 22625.753} C_VEL
LIN {X 0,Y 487.068,Z 954.804,A -85,B 0,C 180,E1 22624.015,E2 22624.015} C_VEL
LIN {X 0,Y 482.433,Z 973.69,A -85,B 0,C 180,E1 22621.765,E2 22621.765} C_VEL
LIN {X 0,Y 478.672,Z 988.961,A -85,B 0,C 180,E1 22619.66,E2 22619.66} C_VEL
LIN {X 0,Y 474.792,Z 1005.322,A -85,B 0,C 180,E1 22617.058,E2 22617.058} C_VEL
LIN {X 0,Y 471.865,Z 1018.2,A -85,B 0,C 180,E1 22614.673,E2 22614.673} C_VEL
LIN {X 0,Y 469.182,Z 1031.211,A -85,B 0,C 180,E1 22611.898,E2 22611.898} C_VEL
LIN {X 0,Y 467.244,Z 1041.71,A -85,B 0,C 180,E1 22609.242,E2 22609.242} C_VEL
LIN {X 0,Y 465.744,Z 1051.561,A -85,B 0,C 180,E1 22606.331,E2 22606.331} C_VEL
LIN {X 0,Y 464.78,Z 1059.433,A -85,B 0,C 180,E1 22603.435,E2 22603.435} C_VEL
LIN {X 0,Y 464.274,Z 1065.294,A -85,B 0,C 180,E1 22600.799,E2 22600.799} C_VEL
LIN {X 0,Y 463.989,Z 1070.518,A -85,B 0,C 180,E1 22597.678,E2 22597.678} C_VEL
LIN {X 0,Y 463.943,Z 1073.39,A -85,B 0,C 180,E1 22595.193,E2 22595.193} C_VEL
LIN {X 0,Y 463.933,Z 1075.237,A -85,B 0,C 180,E1 22592.594,E2 22592.594} C_VEL
LIN {X 0,Y 463.933,Z 1075.821,A -85,B 0,C 180,E1 22589.63,E2 22589.63} C_VEL
LIN {X 0,Y 463.938,Z 1074.979,A -85,B 0,C 180,E1 22587.035,E2 22587.035} C_VEL
LIN {X 0,Y 463.945,Z 1073.072,A -85,B 0,C 180,E1 22584.559,E2 22584.559} C_VEL
LIN {X 0,Y 464.051,Z 1069.098,A -85,B 0,C 180,E1 22581.45,E2 22581.45} C_VEL
LIN {X 0,Y 464.326,Z 1064.288,A -85,B 0,C 180,E1 22578.825,E2 22578.825} C_VEL
LIN {X 0,Y 464.87,Z 1058.203,A -85,B 0,C 180,E1 22576.187,E2 22576.187} C_VEL
LIN {X 0,Y 465.933,Z 1049.446,A -85,B 0,C 180,E1 22573.159,E2 22573.159} C_VEL
LIN {X 0,Y 467.275,Z 1040.658,A -85,B 0,C 180,E1 22570.63,E2 22570.63} C_VEL
LIN {X 0,Y 469.428,Z 1028.73,A -85,B 0,C 180,E1 22567.719,E2 22567.719} C_VEL
LIN {X 0,Y 471.748,Z 1017.173,A -85,B 0,C 180,E1 22565.32,E2 22565.32} C_VEL
LIN {X 0,Y 474.803,Z 1003.351,A -85,B 0,C 180,E1 22562.808,E2 22562.808} C_VEL
LIN {X 0,Y 478.289,Z 987.945,A -85,B 0,C 180,E1 22560.421,E2 22560.421} C_VEL
LIN {X 0,Y 482.157,Z 971.697,A -85,B 0,C 180,E1 22558.214,E2 22558.214} C_VEL
LIN {X 0,Y 486.44,Z 953.32,A -85,B 0,C 180,E1 22556.077,E2 22556.077} C_VEL
LIN {X 0,Y 490.566,Z 935.499,A -85,B 0,C 180,E1 22554.271,E2 22554.271} C_VEL
LIN {X 0,Y 495.107,Z 914.975,A -85,B 0,C 180,E1 22552.491,E2 22552.491} C_VEL
LIN {X 0,Y 499.039,Z 896.208,A -85,B 0,C 180,E1 22551.087,E2 22551.087} C_VEL
LIN {X 0,Y 503.431,Z 873.57,A -85,B 0,C 180,E1 22549.648,E2 22549.648} C_VEL
LIN {X 0,Y 506.962,Z 853.296,A -85,B 0,C 180,E1 22548.569,E2 22548.569} C_VEL
LIN {X 0,Y 510.531,Z 830.393,A -85,B 0,C 180,E1 22547.549,E2 22547.549} C_VEL
LIN {X 0,Y 513.436,Z 807.939,A -85,B 0,C 180,E1 22546.759,E2 22546.759} C_VEL
LIN {X 0,Y 515.735,Z 786.861,A -85,B 0,C 180,E1 22546.17,E2 22546.17} C_VEL
LIN {X 0,Y 517.743,Z 760.82,A -85,B 0,C 180,E1 22545.634,E2 22545.634} C_VEL
LIN {X 0,Y 526.529,Z 534.34,A -85,B 0,C 180,E1 22542.244,E2 22542.244} C_VEL
LIN {X 0,Y 529.359,Z 459.98,A -85,B 0,C 180,E1 22541.116,E2 22541.116} C_VEL
LIN {X 0,Y 517.246,Z 438.875,A -85,B 0,C 180,E1 22539.172,E2 22539.172} C_VEL
LIN {X 0,Y 505.333,Z 419.769,A -85,B 0,C 180,E1 22537.121,E2 22537.121} C_VEL
LIN {X 0,Y 493.247,Z 401.767,A -85,B 0,C 180,E1 22534.866,E2 22534.866} C_VEL
LIN {X 0,Y 483.322,Z 388.058,A -85,B 0,C 180,E1 22532.857,E2 22532.857} C_VEL
LIN {X 0,Y 478.844,Z 382.015,A -85,B 0,C 180,E1 22531.891,E2 22531.891} C_VEL
LIN {X 0,Y 471.574,Z 372.628,A -85,B 0,C 180,E1 22530.237,E2 22530.237} C_VEL
LIN {X 0,Y 468.529,Z 368.452,A -85,B 0,C 180,E1 22529.498,E2 22529.498} C_VEL
LIN {X 0,Y 466.189,Z 363.557,A -85,B 0,C 180,E1 22528.155,E2 22528.155} C_VEL
LIN {X 0,Y 466.121,Z 363.144,A -85,B 0,C 180,E1 22528.02,E2 22528.02} C_VEL
LIN {X 0,Y 466.153,Z 363.146,A -85,B 0,C 180,E1 22524.455,E2 22524.455} C_VEL
LIN {X 0,Y 466.149,Z 363.166,A -85,B 0,C 180,E1 22520.991,E2 22520.991} C_VEL
LIN {X 0,Y 466.118,Z 363.156,A -85,B 0,C 180,E1 22517.477,E2 22517.477} C_VEL
LIN {X 0,Y 466.118,Z 363.139,A -85,B 0,C 180,E1 22513.775,E2 22513.775} C_VEL
LIN {X 0,Y 466.154,Z 363.134,A -85,B 0,C 180,E1 22510.255,E2 22510.255} C_VEL
LIN {X 0,Y 466.161,Z 363.165,A -85,B 0,C 180,E1 22506.651,E2 22506.651} C_VEL
LIN {X 0,Y 466.121,Z 363.148,A -85,B 0,C 180,E1 22503.074,E2 22503.074} C_VEL
LIN {X 0,Y 466.118,Z 363.132,A -85,B 0,C 180,E1 22499.508,E2 22499.508} C_VEL
LIN {X 0,Y 466.151,Z 363.159,A -85,B 0,C 180,E1 22495.941,E2 22495.941} C_VEL
LIN {X 0,Y 466.18,Z 363.151,A -85,B 0,C 180,E1 22492.234,E2 22492.234} C_VEL
LIN {X 0,Y 466.133,Z 363.13,A -85,B 0,C 180,E1 22488.608,E2 22488.608} C_VEL
LIN {X 0,Y 466.118,Z 363.15,A -85,B 0,C 180,E1 22485.083,E2 22485.083} C_VEL
LIN {X 0,Y 466.138,Z 363.169,A -85,B 0,C 180,E1 22481.462,E2 22481.462} C_VEL
LIN {X 0,Y 466.176,Z 363.143,A -85,B 0,C 180,E1 22477.821,E2 22477.821} C_VEL
LIN {X 0,Y 466.149,Z 363.136,A -85,B 0,C 180,E1 22474.187,E2 22474.187} C_VEL
LIN {X 0,Y 466.121,Z 363.141,A -85,B 0,C 180,E1 22470.719,E2 22470.719} C_VEL
LIN {X 0,Y 466.145,Z 363.332,A -85,B 0,C 180,E1 22468.738,E2 22468.738} C_VEL
LIN {X 0,Y 467.136,Z 366.173,A -85,B 0,C 180,E1 22468.443,E2 22468.443} C_VEL
LIN {X 0,Y 469.659,Z 368.809,A -85,B 0,C 180,E1 22467.843,E2 22467.843} C_VEL
LIN {X 0,Y 471.092,Z 369.9,A -85,B 0,C 180,E1 22467.521,E2 22467.521} C_VEL
LIN {X 0,Y 473.328,Z 373.522,A -85,B 0,C 180,E1 22466.974,E2 22466.974} C_VEL
LIN {X 0,Y 476.108,Z 376.165,A -85,B 0,C 180,E1 22466.364,E2 22466.364} C_VEL
LIN {X 0,Y 479.193,Z 380.342,A -85,B 0,C 180,E1 22465.673,E2 22465.673} C_VEL
LIN {X 0,Y 481.043,Z 382.367,A -85,B 0,C 180,E1 22465.282,E2 22465.282} C_VEL
LIN {X 0,Y 485.99,Z 388.713,A -85,B 0,C 180,E1 22464.245,E2 22464.245} C_VEL
LIN {X 0,Y 490.95,Z 395.022,A -85,B 0,C 180,E1 22463.254,E2 22463.254} C_VEL
LIN {X 0,Y 501.016,Z 408.196,A -85,B 0,C 180,E1 22461.361,E2 22461.361} C_VEL
LIN {X 0,Y 513.708,Z 425.991,A -85,B 0,C 180,E1 22459.156,E2 22459.156} C_VEL
LIN {X 0,Y 523.344,Z 440.79,A -85,B 0,C 180,E1 22457.589,E2 22457.589} C_VEL
LIN {X 0,Y 529.658,Z 451.856,A -85,B 0,C 180,E1 22456.591,E2 22456.591} C_VEL
LIN {X 0,Y 519.872,Z 701.036,A -85,B 0,C 180,E1 22452.882,E2 22452.882} C_VEL
LIN {X 0,Y 517.888,Z 747.099,A -85,B 0,C 180,E1 22452.166,E2 22452.166} C_VEL
LIN {X 0,Y 515.883,Z 771.168,A -85,B 0,C 180,E1 22451.612,E2 22451.612} C_VEL
LIN {X 0,Y 513.349,Z 795.051,A -85,B 0,C 180,E1 22450.888,E2 22450.888} C_VEL
LIN {X 0,Y 510.224,Z 818.004,A -85,B 0,C 180,E1 22449.982,E2 22449.982} C_VEL
LIN {X 0,Y 506.989,Z 838.853,A -85,B 0,C 180,E1 22448.986,E2 22448.986} C_VEL
LIN {X 0,Y 502.974,Z 861.197,A -85,B 0,C 180,E1 22447.701,E2 22447.701} C_VEL
LIN {X 0,Y 499.279,Z 879.973,A -85,B 0,C 180,E1 22446.426,E2 22446.426} C_VEL
LIN {X 0,Y 494.747,Z 901.22,A -85,B 0,C 180,E1 22444.745,E2 22444.745} C_VEL
LIN {X 0,Y 490.679,Z 918.969,A -85,B 0,C 180,E1 22443.101,E2 22443.101} C_VEL
LIN {X 0,Y 486.319,Z 937.478,A -85,B 0,C 180,E1 22441.137,E2 22441.137} C_VEL
LIN {X 0,Y 482.171,Z 954.403,A -85,B 0,C 180,E1 22439.029,E2 22439.029} C_VEL
LIN {X 0,Y 478.249,Z 970.673,A -85,B 0,C 180,E1 22436.712,E2 22436.712} C_VEL
LIN {X 0,Y 474.711,Z 985.357,A -85,B 0,C 180,E1 22434.251,E2 22434.251} C_VEL
LIN {X 0,Y 473.68,Z 989.946,A -85,B 0,C 180,E1 22433.424,E2 22433.424} C_VEL
LIN {X 0,Y 471.804,Z 994.228,A -85,B 0,C 180,E1 22432.672,E2 22432.672} C_VEL
LIN {X 0,Y 463.475,Z 1005.134,A -85,B 0,C 180,E1 22430.682,E2 22430.682} C_VEL
LIN {X 0,Y 462.054,Z 1008.223,A -85,B 0,C 180,E1 22429.972,E2 22429.972} C_VEL
LIN {X 0,Y 459.978,Z 1018.321,A -85,B 0,C 180,E1 22427.326,E2 22427.326} C_VEL
LIN {X 0,Y 458.303,Z 1027.843,A -85,B 0,C 180,E1 22424.402,E2 22424.402} C_VEL
LIN {X 0,Y 457.168,Z 1035.458,A -85,B 0,C 180,E1 22421.48,E2 22421.48} C_VEL
LIN {X 0,Y 456.528,Z 1041.112,A -85,B 0,C 180,E1 22418.819,E2 22418.819} C_VEL
LIN {X 0,Y 456.122,Z 1046.237,A -85,B 0,C 180,E1 22415.59,E2 22415.59} C_VEL
LIN {X 0,Y 455.993,Z 1049.024,A -85,B 0,C 180,E1 22413.017,E2 22413.017} C_VEL
LIN {X 0,Y 455.957,Z 1050.829,A -85,B 0,C 180,E1 22410.251,E2 22410.251} C_VEL
LIN {X 0,Y 455.936,Z 1051.23,A -85,B 0,C 180,E1 22407.235,E2 22407.235} C_VEL
LIN {X 0,Y 455.961,Z 1050.407,A -85,B 0,C 180,E1 22404.715,E2 22404.715} C_VEL
LIN {X 0,Y 456.03,Z 1048.428,A -85,B 0,C 180,E1 22402.06,E2 22402.06} C_VEL
LIN {X 0,Y 456.268,Z 1044.431,A -85,B 0,C 180,E1 22398.881,E2 22398.881} C_VEL
LIN {X 0,Y 456.698,Z 1039.948,A -85,B 0,C 180,E1 22396.323,E2 22396.323} C_VEL
LIN {X 0,Y 457.565,Z 1033.418,A -85,B 0,C 180,E1 22393.365,E2 22393.365} C_VEL
LIN {X 0,Y 458.928,Z 1025.023,A -85,B 0,C 180,E1 22390.395,E2 22390.395} C_VEL
LIN {X 0,Y 460.826,Z 1015.455,A -85,B 0,C 180,E1 22387.55,E2 22387.55} C_VEL
LIN {X 0,Y 463.387,Z 1003.91,A -85,B 0,C 180,E1 22384.705,E2 22384.705} C_VEL
LIN {X 0,Y 466.368,Z 991.804,A -85,B 0,C 180,E1 22382.135,E2 22382.135} C_VEL
LIN {X 0,Y 470.149,Z 977.028,A -85,B 0,C 180,E1 22379.467,E2 22379.467} C_VEL
LIN {X 0,Y 473.82,Z 963.193,A -85,B 0,C 180,E1 22377.301,E2 22377.301} C_VEL
LIN {X 0,Y 478.625,Z 945.105,A -85,B 0,C 180,E1 22374.862,E2 22374.862} C_VEL
LIN {X 0,Y 482.842,Z 928.989,A -85,B 0,C 180,E1 22372.988,E2 22372.988} C_VEL
LIN {X 0,Y 487.97,Z 908.659,A -85,B 0,C 180,E1 22370.951,E2 22370.951} C_VEL
LIN {X 0,Y 492.318,Z 890.419,A -85,B 0,C 180,E1 22369.388,E2 22369.388} C_VEL
LIN {X 0,Y 497.275,Z 868.075,A -85,B 0,C 180,E1 22367.754,E2 22367.754} C_VEL
LIN {X 0,Y 501.059,Z 849.129,A -85,B 0,C 180,E1 22366.584,E2 22366.584} C_VEL
LIN {X 0,Y 505.057,Z 827.238,A -85,B 0,C 180,E1 22365.434,E2 22365.434} C_VEL
LIN {X 0,Y 508.423,Z 805.036,A -85,B 0,C 180,E1 22364.488,E2 22364.488} C_VEL
LIN {X 0,Y 511.082,Z 784.633,A -85,B 0,C 180,E1 22363.777,E2 22363.777} C_VEL
LIN {X 0,Y 513.702,Z 759.184,A -85,B 0,C 180,E1 22363.095,E2 22363.095} C_VEL
LIN {X 0,Y 515.224,Z 737.466,A -85,B 0,C 180,E1 22362.672,E2 22362.672} C_VEL
LIN {X 0,Y 525.825,Z 490.776,A -85,B 0,C 180,E1 22358.948,E2 22358.948} C_VEL
LIN {X 0,Y 527.226,Z 456.518,A -85,B 0,C 180,E1 22358.415,E2 22358.415} C_VEL
LIN {X 0,Y 518.4,Z 442.163,A -85,B 0,C 180,E1 22356.894,E2 22356.894} C_VEL
LIN {X 0,Y 506.621,Z 425.172,A -85,B 0,C 180,E1 22354.743,E2 22354.743} C_VEL
LIN {X 0,Y 495.272,Z 409.956,A -85,B 0,C 180,E1 22352.481,E2 22352.481} C_VEL
LIN {X 0,Y 486.502,Z 398.885,A -85,B 0,C 180,E1 22350.576,E2 22350.576} C_VEL
LIN {X 0,Y 482.516,Z 393.936,A -85,B 0,C 180,E1 22349.653,E2 22349.653} C_VEL
LIN {X 0,Y 478.206,Z 388.608,A -85,B 0,C 180,E1 22348.609,E2 22348.609} C_VEL
LIN {X 0,Y 474.75,Z 384.598,A -85,B 0,C 180,E1 22347.74,E2 22347.74} C_VEL
LIN {X 0,Y 473.508,Z 382.871,A -85,B 0,C 180,E1 22347.409,E2 22347.409} C_VEL
LIN {X 0,Y 470.244,Z 379.565,A -85,B 0,C 180,E1 22346.555,E2 22346.555} C_VEL
LIN {X 0,Y 468.592,Z 376.914,A -85,B 0,C 180,E1 22346.076,E2 22346.076} C_VEL
LIN {X 0,Y 465.331,Z 374.096,A -85,B 0,C 180,E1 22345.18,E2 22345.18} C_VEL
LIN {X 0,Y 463.531,Z 370.718,A -85,B 0,C 180,E1 22344.603,E2 22344.603} C_VEL
LIN {X 0,Y 460.185,Z 368.505,A -85,B 0,C 180,E1 22343.633,E2 22343.633} C_VEL
LIN {X 0,Y 458.546,Z 365.742,A -85,B 0,C 180,E1 22343.076,E2 22343.076} C_VEL
LIN {X 0,Y 458.182,Z 364.15,A -85,B 0,C 180,E1 22342.896,E2 22342.896} C_VEL
LIN {X 0,Y 458.186,Z 364.15,A -85,B 0,C 180,E1 22339.24,E2 22339.24} C_VEL
LIN {X 0,Y 458.219,Z 364.153,A -85,B 0,C 180,E1 22335.699,E2 22335.699} C_VEL
LIN {X 0,Y 458.221,Z 364.153,A -85,B 0,C 180,E1 22332.092,E2 22332.092} C_VEL
LIN {X 0,Y 458.186,Z 364.146,A -85,B 0,C 180,E1 22328.534,E2 22328.534} C_VEL
LIN {X 0,Y 458.178,Z 364.137,A -85,B 0,C 180,E1 22324.882,E2 22324.882} C_VEL
LIN {X 0,Y 458.197,Z 364.129,A -85,B 0,C 180,E1 22321.25,E2 22321.25} C_VEL
LIN {X 0,Y 458.224,Z 364.129,A -85,B 0,C 180,E1 22317.749,E2 22317.749} C_VEL
LIN {X 0,Y 458.194,Z 364.142,A -85,B 0,C 180,E1 22314.113,E2 22314.113} C_VEL
LIN {X 0,Y 458.18,Z 364.159,A -85,B 0,C 180,E1 22310.541,E2 22310.541} C_VEL
LIN {X 0,Y 458.191,Z 364.153,A -85,B 0,C 180,E1 22306.882,E2 22306.882} C_VEL
LIN {X 0,Y 458.226,Z 364.135,A -85,B 0,C 180,E1 22303.323,E2 22303.323} C_VEL
LIN {X 0,Y 458.205,Z 364.131,A -85,B 0,C 180,E1 22299.698,E2 22299.698} C_VEL
LIN {X 0,Y 458.177,Z 364.133,A -85,B 0,C 180,E1 22296.188,E2 22296.188} C_VEL
LIN {X 0,Y 458.216,Z 364.355,A -85,B 0,C 180,E1 22295.917,E2 22295.917} C_VEL
LIN {X 0,Y 459.577,Z 367.733,A -85,B 0,C 180,E1 22294.896,E2 22294.896} C_VEL
LIN {X 0,Y 462.088,Z 370.554,A -85,B 0,C 180,E1 22294.115,E2 22294.115} C_VEL
LIN {X 0,Y 465.638,Z 374.677,A -85,B 0,C 180,E1 22293.058,E2 22293.058} C_VEL
LIN {X 0,Y 469.986,Z 380.296,A -85,B 0,C 180,E1 22291.816,E2 22291.816} C_VEL
LIN {X 0,Y 472.027,Z 382.917,A -85,B 0,C 180,E1 22291.259,E2 22291.259} C_VEL
LIN {X 0,Y 479.259,Z 392.183,A -85,B 0,C 180,E1 22289.398,E2 22289.398} C_VEL
LIN {X 0,Y 484.358,Z 399.161,A -85,B 0,C 180,E1 22288.167,E2 22288.167} C_VEL
LIN {X 0,Y 490.134,Z 406.894,A -85,B 0,C 180,E1 22286.857,E2 22286.857} C_VEL
LIN {X 0,Y 501.797,Z 423.689,A -85,B 0,C 180,E1 22284.402,E2 22284.402} C_VEL
LIN {X 0,Y 513.715,Z 442.294,A -85,B 0,C 180,E1 22282.114,E2 22282.114} C_VEL
LIN {X 0,Y 525.097,Z 461.488,A -85,B 0,C 180,E1 22280.098,E2 22280.098} C_VEL
LIN {X 0,Y 527.168,Z 465.478,A -85,B 0,C 180,E1 22279.739,E2 22279.739} C_VEL
LIN {X 0,Y 516.596,Z 712.931,A -85,B 0,C 180,E1 22276.011,E2 22276.011} C_VEL
LIN {X 0,Y 514.201,Z 765.76,A -85,B 0,C 180,E1 22275.188,E2 22275.188} C_VEL
LIN {X 0,Y 511.93,Z 790.227,A -85,B 0,C 180,E1 22274.645,E2 22274.645} C_VEL
LIN {X 0,Y 509.45,Z 811,A -85,B 0,C 180,E1 22274.043,E2 22274.043} C_VEL
LIN {X 0,Y 505.908,Z 835.192,A -85,B 0,C 180,E1 22273.145,E2 22273.145} C_VEL
LIN {X 0,Y 502.614,Z 854.609,A -85,B 0,C 180,E1 22272.253,E2 22272.253} C_VEL
LIN {X 0,Y 498.359,Z 877.126,A -85,B 0,C 180,E1 22271.027,E2 22271.027} C_VEL
LIN {X 0,Y 493.82,Z 898.296,A -85,B 0,C 180,E1 22269.629,E2 22269.629} C_VEL
LIN {X 0,Y 489.154,Z 918.858,A -85,B 0,C 180,E1 22268.047,E2 22268.047} C_VEL
LIN {X 0,Y 484.379,Z 938.312,A -85,B 0,C 180,E1 22266.276,E2 22266.276} C_VEL
LIN {X 0,Y 480.121,Z 955.271,A -85,B 0,C 180,E1 22264.504,E2 22264.504} C_VEL
LIN {X 0,Y 475.397,Z 973.705,A -85,B 0,C 180,E1 22262.272,E2 22262.272} C_VEL
LIN {X 0,Y 471.522,Z 988.749,A -85,B 0,C 180,E1 22260.17,E2 22260.17} C_VEL
LIN {X 0,Y 467.427,Z 1005.18,A -85,B 0,C 180,E1 22257.52,E2 22257.52} C_VEL
LIN {X 0,Y 464.352,Z 1018.05,A -85,B 0,C 180,E1 22255.1,E2 22255.1} C_VEL
LIN {X 0,Y 461.523,Z 1031.047,A -85,B 0,C 180,E1 22252.28,E2 22252.28} C_VEL
LIN {X 0,Y 459.443,Z 1041.649,A -85,B 0,C 180,E1 22249.551,E2 22249.551} C_VEL
LIN {X 0,Y 457.874,Z 1051.37,A -85,B 0,C 180,E1 22246.623,E2 22246.623} C_VEL
LIN {X 0,Y 456.835,Z 1059.329,A -85,B 0,C 180,E1 22243.639,E2 22243.639} C_VEL
LIN {X 0,Y 456.284,Z 1065.362,A -85,B 0,C 180,E1 22240.863,E2 22240.863} C_VEL
LIN {X 0,Y 455.995,Z 1070.318,A -85,B 0,C 180,E1 22237.814,E2 22237.814} C_VEL
LIN {X 0,Y 455.944,Z 1073.186,A -85,B 0,C 180,E1 22235.285,E2 22235.285} C_VEL
LIN {X 0,Y 455.935,Z 1075.029,A -85,B 0,C 180,E1 22232.64,E2 22232.64} C_VEL
LIN {X 0,Y 455.936,Z 1075.605,A -85,B 0,C 180,E1 22229.623,E2 22229.623} C_VEL
LIN {X 0,Y 455.94,Z 1074.759,A -85,B 0,C 180,E1 22226.983,E2 22226.983} C_VEL
LIN {X 0,Y 455.947,Z 1072.847,A -85,B 0,C 180,E1 22224.463,E2 22224.463} C_VEL
LIN {X 0,Y 456.052,Z 1069.07,A -85,B 0,C 180,E1 22221.424,E2 22221.424} C_VEL
LIN {X 0,Y 456.354,Z 1064.045,A -85,B 0,C 180,E1 22218.627,E2 22218.627} C_VEL
LIN {X 0,Y 456.974,Z 1057.644,A -85,B 0,C 180,E1 22215.814,E2 22215.814} C_VEL
LIN {X 0,Y 458.072,Z 1049.184,A -85,B 0,C 180,E1 22212.862,E2 22212.862} C_VEL
LIN {X 0,Y 459.49,Z 1040.389,A -85,B 0,C 180,E1 22210.288,E2 22210.288} C_VEL
LIN {X 0,Y 461.815,Z 1028.187,A -85,B 0,C 180,E1 22207.272,E2 22207.272} C_VEL
LIN {X 0,Y 464.219,Z 1016.881,A -85,B 0,C 180,E1 22204.892,E2 22204.892} C_VEL
LIN {X 0,Y 467.596,Z 1002.267,A -85,B 0,C 180,E1 22202.215,E2 22202.215} C_VEL
LIN {X 0,Y 471.059,Z 987.73,A -85,B 0,C 180,E1 22199.938,E2 22199.938} C_VEL
LIN {X 0,Y 475.213,Z 971.011,A -85,B 0,C 180,E1 22197.64,E2 22197.64} C_VEL
LIN {X 0,Y 479.52,Z 953.243,A -85,B 0,C 180,E1 22195.555,E2 22195.555} C_VEL
LIN {X 0,Y 483.735,Z 935.751,A -85,B 0,C 180,E1 22193.76,E2 22193.76} C_VEL
LIN {X 0,Y 488.441,Z 915.324,A -85,B 0,C 180,E1 22191.962,E2 22191.962} C_VEL
LIN {X 0,Y 492.504,Z 896.616,A -85,B 0,C 180,E1 22190.546,E2 22190.546} C_VEL
LIN {X 0,Y 497.11,Z 873.76,A -85,B 0,C 180,E1 22189.075,E2 22189.075} C_VEL
LIN {X 0,Y 500.682,Z 853.949,A -85,B 0,C 180,E1 22188.009,E2 22188.009} C_VEL
LIN {X 0,Y 504.312,Z 831.603,A -85,B 0,C 180,E1 22186.997,E2 22186.997} C_VEL
LIN {X 0,Y 507.469,Z 808.093,A -85,B 0,C 180,E1 22186.158,E2 22186.158} C_VEL
LIN {X 0,Y 509.804,Z 787.373,A -85,B 0,C 180,E1 22185.572,E2 22185.572} C_VEL
LIN {X 0,Y 511.932,Z 760.897,A -85,B 0,C 180,E1 22185.02,E2 22185.02} C_VEL
LIN {X 0,Y 520.999,Z 535.801,A -85,B 0,C 180,E1 22181.624,E2 22181.624} C_VEL
LIN {X 0,Y 523.883,Z 463.407,A -85,B 0,C 180,E1 22180.52,E2 22180.52} C_VEL
LIN {X 0,Y 511.785,Z 442.286,A -85,B 0,C 180,E1 22178.518,E2 22178.518} C_VEL
LIN {X 0,Y 500.842,Z 424.786,A -85,B 0,C 180,E1 22176.579,E2 22176.579} C_VEL
LIN {X 0,Y 489.825,Z 408.153,A -85,B 0,C 180,E1 22174.469,E2 22174.469} C_VEL
LIN {X 0,Y 479.895,Z 394.334,A -85,B 0,C 180,E1 22172.412,E2 22172.412} C_VEL
LIN {X 0,Y 475.36,Z 388.159,A -85,B 0,C 180,E1 22171.408,E2 22171.408} C_VEL
LIN {X 0,Y 468.654,Z 379.399,A -85,B 0,C 180,E1 22169.845,E2 22169.845} C_VEL
LIN {X 0,Y 464.766,Z 374.244,A -85,B 0,C 180,E1 22168.881,E2 22168.881} C_VEL
LIN {X 0,Y 461.291,Z 369.861,A -85,B 0,C 180,E1 22167.988,E2 22167.988} C_VEL
LIN {X 0,Y 459.51,Z 367.643,A -85,B 0,C 180,E1 22167.472,E2 22167.472} C_VEL
LIN {X 0,Y 458.209,Z 364.129,A -85,B 0,C 180,E1 22166.434,E2 22166.434} C_VEL
LIN {X 0,Y 458.237,Z 364.121,A -85,B 0,C 180,E1 22162.72,E2 22162.72} C_VEL
LIN {X 0,Y 458.195,Z 364.124,A -85,B 0,C 180,E1 22159.107,E2 22159.107} C_VEL
LIN {X 0,Y 458.177,Z 364.139,A -85,B 0,C 180,E1 22155.571,E2 22155.571} C_VEL
LIN {X 0,Y 458.196,Z 364.158,A -85,B 0,C 180,E1 22151.965,E2 22151.965} C_VEL
LIN {X 0,Y 458.225,Z 364.127,A -85,B 0,C 180,E1 22148.28,E2 22148.28} C_VEL
LIN {X 0,Y 458.202,Z 364.12,A -85,B 0,C 180,E1 22144.757,E2 22144.757} C_VEL
LIN {X 0,Y 458.182,Z 364.151,A -85,B 0,C 180,E1 22141.125,E2 22141.125} C_VEL
LIN {X 0,Y 458.179,Z 364.147,A -85,B 0,C 180,E1 22137.373,E2 22137.373} C_VEL
LIN {X 0,Y 458.196,Z 364.119,A -85,B 0,C 180,E1 22133.736,E2 22133.736} C_VEL
LIN {X 0,Y 458.227,Z 364.131,A -85,B 0,C 180,E1 22130.2,E2 22130.2} C_VEL
LIN {X 0,Y 458.205,Z 364.154,A -85,B 0,C 180,E1 22126.497,E2 22126.497} C_VEL
LIN {X 0,Y 458.18,Z 364.131,A -85,B 0,C 180,E1 22122.911,E2 22122.911} C_VEL
LIN {X 0,Y 458.187,Z 364.124,A -85,B 0,C 180,E1 22119.297,E2 22119.297} C_VEL
LIN {X 0,Y 458.228,Z 364.132,A -85,B 0,C 180,E1 22115.78,E2 22115.78} C_VEL
LIN {X 0,Y 458.228,Z 364.144,A -85,B 0,C 180,E1 22112.021,E2 22112.021} C_VEL
LIN {X 0,Y 458.211,Z 364.286,A -85,B 0,C 180,E1 22110.474,E2 22110.474} C_VEL
LIN {X 0,Y 459.283,Z 367.238,A -85,B 0,C 180,E1 22110.132,E2 22110.132} C_VEL
LIN {X 0,Y 462.015,Z 369.995,A -85,B 0,C 180,E1 22109.43,E2 22109.43} C_VEL
LIN {X 0,Y 463.272,Z 370.893,A -85,B 0,C 180,E1 22109.127,E2 22109.127} C_VEL
LIN {X 0,Y 465.505,Z 374.546,A -85,B 0,C 180,E1 22108.536,E2 22108.536} C_VEL
LIN {X 0,Y 468.396,Z 377.252,A -85,B 0,C 180,E1 22107.854,E2 22107.854} C_VEL
LIN {X 0,Y 471.287,Z 381.231,A -85,B 0,C 180,E1 22107.157,E2 22107.157} C_VEL
LIN {X 0,Y 473.371,Z 383.378,A -85,B 0,C 180,E1 22106.688,E2 22106.688} C_VEL
LIN {X 0,Y 476.936,Z 387.841,A -85,B 0,C 180,E1 22105.888,E2 22105.888} C_VEL
LIN {X 0,Y 483.044,Z 395.643,A -85,B 0,C 180,E1 22104.578,E2 22104.578} C_VEL
LIN {X 0,Y 490.401,Z 405.035,A -85,B 0,C 180,E1 22103.097,E2 22103.097} C_VEL
LIN {X 0,Y 502.827,Z 421.982,A -85,B 0,C 180,E1 22100.776,E2 22100.776} C_VEL
LIN {X 0,Y 514.636,Z 439.254,A -85,B 0,C 180,E1 22098.748,E2 22098.748} C_VEL
LIN {X 0,Y 523.263,Z 453.508,A -85,B 0,C 180,E1 22097.34,E2 22097.34} C_VEL
LIN {X 0,Y 524.166,Z 455.48,A -85,B 0,C 180,E1 22097.188,E2 22097.188} C_VEL
LIN {X 0,Y 513.961,Z 706.192,A -85,B 0,C 180,E1 22093.428,E2 22093.428} C_VEL
LIN {X 0,Y 512.058,Z 747.8,A -85,B 0,C 180,E1 22092.771,E2 22092.771} C_VEL
LIN {X 0,Y 510.005,Z 771.636,A -85,B 0,C 180,E1 22092.217,E2 22092.217} C_VEL
LIN {X 0,Y 507.431,Z 795.134,A -85,B 0,C 180,E1 22091.501,E2 22091.501} C_VEL
LIN {X 0,Y 504.175,Z 818.329,A -85,B 0,C 180,E1 22090.579,E2 22090.579} C_VEL
LIN {X 0,Y 500.793,Z 839.443,A -85,B 0,C 180,E1 22089.562,E2 22089.562} C_VEL
LIN {X 0,Y 496.611,Z 861.877,A -85,B 0,C 180,E1 22088.257,E2 22088.257} C_VEL
LIN {X 0,Y 492.66,Z 881.26,A -85,B 0,C 180,E1 22086.924,E2 22086.924} C_VEL
LIN {X 0,Y 487.817,Z 902.979,A -85,B 0,C 180,E1 22085.168,E2 22085.168} C_VEL
LIN {X 0,Y 483.789,Z 919.932,A -85,B 0,C 180,E1 22083.571,E2 22083.571} C_VEL
LIN {X 0,Y 479.098,Z 938.966,A -85,B 0,C 180,E1 22081.506,E2 22081.506} C_VEL
LIN {X 0,Y 475.07,Z 954.781,A -85,B 0,C 180,E1 22079.505,E2 22079.505} C_VEL
LIN {X 0,Y 470.99,Z 971.03,A -85,B 0,C 180,E1 22077.157,E2 22077.157} C_VEL
LIN {X 0,Y 467.289,Z 985.698,A -85,B 0,C 180,E1 22074.661,E2 22074.661} C_VEL
LIN {X 0,Y 464.096,Z 999.223,A -85,B 0,C 180,E1 22072.017,E2 22072.017} C_VEL
LIN {X 0,Y 462.054,Z 1008.223,A -85,B 0,C 180,E1 22069.972,E2 22069.972} C_VEL
LIN {X 0,Y 460.335,Z 1011.752,A -85,B 0,C 180,E1 22069.138,E2 22069.138} C_VEL
LIN {X 0,Y 452.501,Z 1020.938,A -85,B 0,C 180,E1 22066.94,E2 22066.94} C_VEL
LIN {X 0,Y 451.27,Z 1023.48,A -85,B 0,C 180,E1 22066.176,E2 22066.176} C_VEL
LIN {X 0,Y 449.909,Z 1031.245,A -85,B 0,C 180,E1 22063.495,E2 22063.495} C_VEL
LIN {X 0,Y 448.891,Z 1038.635,A -85,B 0,C 180,E1 22060.394,E2 22060.394} C_VEL
LIN {X 0,Y 448.318,Z 1043.981,A -85,B 0,C 180,E1 22057.432,E2 22057.432} C_VEL
LIN {X 0,Y 448.067,Z 1047.8,A -85,B 0,C 180,E1 22054.608,E2 22054.608} C_VEL
LIN {X 0,Y 447.969,Z 1050.386,A -85,B 0,C 180,E1 22051.535,E2 22051.535} C_VEL
LIN {X 0,Y 447.946,Z 1051.365,A -85,B 0,C 180,E1 22048.977,E2 22048.977} C_VEL
LIN {X 0,Y 447.945,Z 1051.286,A -85,B 0,C 180,E1 22046.288,E2 22046.288} C_VEL
LIN {X 0,Y 448.003,Z 1049.625,A -85,B 0,C 180,E1 22043.078,E2 22043.078} C_VEL
LIN {X 0,Y 448.14,Z 1046.892,A -85,B 0,C 180,E1 22040.367,E2 22040.367} C_VEL
LIN {X 0,Y 448.485,Z 1042.782,A -85,B 0,C 180,E1 22037.511,E2 22037.511} C_VEL
LIN {X 0,Y 449.242,Z 1036.576,A -85,B 0,C 180,E1 22034.377,E2 22034.377} C_VEL
LIN {X 0,Y 450.334,Z 1029.744,A -85,B 0,C 180,E1 22031.622,E2 22031.622} C_VEL
LIN {X 0,Y 452.29,Z 1019.684,A -85,B 0,C 180,E1 22028.334,E2 22028.334} C_VEL
LIN {X 0,Y 454.442,Z 1010.029,A -85,B 0,C 180,E1 22025.704,E2 22025.704} C_VEL
LIN {X 0,Y 457.697,Z 996.962,A -85,B 0,C 180,E1 22022.692,E2 22022.692} C_VEL
LIN {X 0,Y 460.846,Z 985.072,A -85,B 0,C 180,E1 22020.351,E2 22020.351} C_VEL
LIN {X 0,Y 465.013,Z 970.007,A -85,B 0,C 180,E1 22017.774,E2 22017.774} C_VEL
LIN {X 0,Y 469.151,Z 954.945,A -85,B 0,C 180,E1 22015.569,E2 22015.569} C_VEL
LIN {X 0,Y 474.018,Z 937.548,A -85,B 0,C 180,E1 22013.348,E2 22013.348} C_VEL
LIN {X 0,Y 478.863,Z 919.276,A -85,B 0,C 180,E1 22011.367,E2 22011.367} C_VEL
LIN {X 0,Y 483.509,Z 901.231,A -85,B 0,C 180,E1 22009.663,E2 22009.663} C_VEL
LIN {X 0,Y 488.483,Z 880.317,A -85,B 0,C 180,E1 22007.983,E2 22007.983} C_VEL
LIN {X 0,Y 492.633,Z 861.423,A -85,B 0,C 180,E1 22006.683,E2 22006.683} C_VEL
LIN {X 0,Y 497.429,Z 837.175,A -85,B 0,C 180,E1 22005.288,E2 22005.288} C_VEL
LIN {X 0,Y 500.903,Z 816.864,A -85,B 0,C 180,E1 22004.32,E2 22004.32} C_VEL
LIN {X 0,Y 504.59,Z 791.469,A -85,B 0,C 180,E1 22003.344,E2 22003.344} C_VEL
LIN {X 0,Y 507.126,Z 769.58,A -85,B 0,C 180,E1 22002.693,E2 22002.693} C_VEL
LIN {X 0,Y 509.367,Z 743.567,A -85,B 0,C 180,E1 22002.123,E2 22002.123} C_VEL
LIN {X 0,Y 514.188,Z 636.015,A -85,B 0,C 180,E1 22000.471,E2 22000.471} C_VEL
LIN {X 0,Y 522.059,Z 460.243,A -85,B 0,C 180,E1 21997.799,E2 21997.799} C_VEL
LIN {X 0,Y 513.94,Z 447.186,A -85,B 0,C 180,E1 21996.364,E2 21996.364} C_VEL
LIN {X 0,Y 502.833,Z 431.077,A -85,B 0,C 180,E1 21994.281,E2 21994.281} C_VEL
LIN {X 0,Y 492.123,Z 416.54,A -85,B 0,C 180,E1 21992.094,E2 21992.094} C_VEL
LIN {X 0,Y 483.349,Z 405.363,A -85,B 0,C 180,E1 21990.144,E2 21990.144} C_VEL
LIN {X 0,Y 479.641,Z 400.723,A -85,B 0,C 180,E1 21989.265,E2 21989.265} C_VEL
LIN {X 0,Y 475.383,Z 395.471,A -85,B 0,C 180,E1 21988.212,E2 21988.212} C_VEL
LIN {X 0,Y 471.694,Z 390.827,A -85,B 0,C 180,E1 21987.25,E2 21987.25} C_VEL
LIN {X 0,Y 467.461,Z 386.141,A -85,B 0,C 180,E1 21986.11,E2 21986.11} C_VEL
LIN {X 0,Y 465.998,Z 384.075,A -85,B 0,C 180,E1 21985.686,E2 21985.686} C_VEL
LIN {X 0,Y 462.725,Z 380.846,A -85,B 0,C 180,E1 21984.751,E2 21984.751} C_VEL
LIN {X 0,Y 461,Z 378.066,A -85,B 0,C 180,E1 21984.201,E2 21984.201} C_VEL
LIN {X 0,Y 457.667,Z 375.328,A -85,B 0,C 180,E1 21983.191,E2 21983.191} C_VEL
LIN {X 0,Y 455.565,Z 371.69,A -85,B 0,C 180,E1 21982.452,E2 21982.452} C_VEL
LIN {X 0,Y 452.317,Z 369.569,A -85,B 0,C 180,E1 21981.392,E2 21981.392} C_VEL
LIN {X 0,Y 450.629,Z 366.764,A -85,B 0,C 180,E1 21980.744,E2 21980.744} C_VEL
LIN {X 0,Y 450.258,Z 365.131,A -85,B 0,C 180,E1 21980.541,E2 21980.541} C_VEL
LIN {X 0,Y 450.24,Z 365.13,A -85,B 0,C 180,E1 21976.913,E2 21976.913} C_VEL
LIN {X 0,Y 450.245,Z 365.125,A -85,B 0,C 180,E1 21973.223,E2 21973.223} C_VEL
LIN {X 0,Y 450.274,Z 365.117,A -85,B 0,C 180,E1 21969.587,E2 21969.587} C_VEL
LIN {X 0,Y 450.281,Z 365.115,A -85,B 0,C 180,E1 21965.991,E2 21965.991} C_VEL
LIN {X 0,Y 450.244,Z 365.128,A -85,B 0,C 180,E1 21962.418,E2 21962.418} C_VEL
LIN {X 0,Y 450.242,Z 365.141,A -85,B 0,C 180,E1 21958.727,E2 21958.727} C_VEL
LIN {X 0,Y 450.254,Z 365.147,A -85,B 0,C 180,E1 21955.031,E2 21955.031} C_VEL
LIN {X 0,Y 450.289,Z 365.128,A -85,B 0,C 180,E1 21951.444,E2 21951.444} C_VEL
LIN {X 0,Y 450.277,Z 365.12,A -85,B 0,C 180,E1 21947.691,E2 21947.691} C_VEL
LIN {X 0,Y 450.242,Z 365.118,A -85,B 0,C 180,E1 21944.148,E2 21944.148} C_VEL
LIN {X 0,Y 450.236,Z 365.118,A -85,B 0,C 180,E1 21940.407,E2 21940.407} C_VEL
LIN {X 0,Y 450.27,Z 365.319,A -85,B 0,C 180,E1 21938.026,E2 21938.026} C_VEL
LIN {X 0,Y 450.835,Z 367.205,A -85,B 0,C 180,E1 21937.506,E2 21937.506} C_VEL
LIN {X 0,Y 452.772,Z 370.012,A -85,B 0,C 180,E1 21936.784,E2 21936.784} C_VEL
LIN {X 0,Y 455.076,Z 371.943,A -85,B 0,C 180,E1 21936.016,E2 21936.016} C_VEL
LIN {X 0,Y 460.359,Z 378.534,A -85,B 0,C 180,E1 21934.288,E2 21934.288} C_VEL
LIN {X 0,Y 464.269,Z 383.156,A -85,B 0,C 180,E1 21933.11,E2 21933.11} C_VEL
LIN {X 0,Y 468.019,Z 387.859,A -85,B 0,C 180,E1 21932.034,E2 21932.034} C_VEL
LIN {X 0,Y 476.867,Z 399.572,A -85,B 0,C 180,E1 21929.682,E2 21929.682} C_VEL
LIN {X 0,Y 485.216,Z 410.905,A -85,B 0,C 180,E1 21927.673,E2 21927.673} C_VEL
LIN {X 0,Y 493.768,Z 423.223,A -85,B 0,C 180,E1 21925.774,E2 21925.774} C_VEL
LIN {X 0,Y 501.974,Z 435.595,A -85,B 0,C 180,E1 21924.082,E2 21924.082} C_VEL
LIN {X 0,Y 512.044,Z 451.745,A -85,B 0,C 180,E1 21922.146,E2 21922.146} C_VEL
LIN {X 0,Y 521.934,Z 468.785,A -85,B 0,C 180,E1 21920.368,E2 21920.368} C_VEL
LIN {X 0,Y 511.106,Z 713.472,A -85,B 0,C 180,E1 21916.657,E2 21916.657} C_VEL
LIN {X 0,Y 508.654,Z 765.631,A -85,B 0,C 180,E1 21915.838,E2 21915.838} C_VEL
LIN {X 0,Y 506.312,Z 790.128,A -85,B 0,C 180,E1 21915.292,E2 21915.292} C_VEL
LIN {X 0,Y 503.745,Z 810.967,A -85,B 0,C 180,E1 21914.685,E2 21914.685} C_VEL
LIN {X 0,Y 500.065,Z 835.287,A -85,B 0,C 180,E1 21913.775,E2 21913.775} C_VEL
LIN {X 0,Y 496.645,Z 854.769,A -85,B 0,C 180,E1 21912.875,E2 21912.875} C_VEL
LIN {X 0,Y 492.202,Z 877.43,A -85,B 0,C 180,E1 21911.628,E2 21911.628} C_VEL
